ACTION A_ResetFault:
// Sadece arızaları temizle
stHMI.stStatus.bFaultActive := FALSE;
stHMI.stStatus.eFaultCode := E_DisconnectorFault.NONE;
stHMI.stStatus.wsStatusText := "";  // Status text'i temizle

// Timer'ları resetle
tonMotionTimeout(IN := FALSE);
tonContactorOn(IN := FALSE);
tonContactorOff(IN := FALSE);
END_ACTION

ACTION A_ResetStatistics:
// Sadece istatistikleri sıfırla
stHMI.stStatistics.dwOnCount := 0;
stHMI.stStatistics.dwOffCount := 0;
stHMI.stStatistics.dwOperationCount := 0;
stHMI.stStatistics.dwTotalFaultCount := 0;
stHMI.stStatistics.dwThermalFaultCount := 0;
stHMI.stStatistics.dwMotionTimeoutCount := 0;
stHMI.stStatistics.dwContactorFaultCount := 0;
stHMI.stStatistics.dwInterlockFaultCount := 0;
stHMI.stStatistics.tMaxOnTransitionTime := T#0S;
stHMI.stStatistics.tMaxOffTransitionTime := T#0S;
stHMI.stStatistics.tLastOnTransitionTime := T#0S;
stHMI.stStatistics.tLastOffTransitionTime := T#0S;
stHMI.stStatistics.bNewOperationFlag := FALSE;

// Bakım sayacını sıfırla ve operasyon limitini yeniden yükle
stHMI.stStatistics.dwRemainingOperations := stHMI.stConfig.dwOperationLimit;
stHMI.stStatistics.bMaintenanceRequired := FALSE;
END_ACTION

ACTION A_StateMachine:
// Önceki durumu sakla
ePositionPrevious := ePosition;

// Interlock kontrolü
IF bInterlock THEN
    bOnRequest := FALSE;
    bOffRequest := FALSE;
END_IF

// Sürekli pozisyon kontrolü
IF bLimitOn AND bLimitOff THEN
    // Her iki limit aktif - arıza
    ePosition := E_DisconnectorPosition.FAULT;
    stHMI.stStatus.eFaultCode := E_DisconnectorFault.BOTH_LIMITS;
END_IF

// Durum makinesi
CASE ePosition OF
    E_DisconnectorPosition.UNDEFINED:
        // Pozisyon belirleme
        IF bLimitOn AND NOT bLimitOff THEN
            ePosition := E_DisconnectorPosition.ON;
        ELSIF bLimitOff AND NOT bLimitOn THEN
            ePosition := E_DisconnectorPosition.OFF;
        ELSE
            // Ara konumda - komut bekle
            IF bOnRequest THEN
                ePosition := E_DisconnectorPosition.TURNING_ON;
                tOperationStartTime := TIME();
            ELSIF bOffRequest THEN
                ePosition := E_DisconnectorPosition.TURNING_OFF;
                tOperationStartTime := TIME();
            END_IF
        END_IF
        
    E_DisconnectorPosition.OFF:
        // OFF konumunda toprak bıçağı kontrolü
        IF stHMI.stConfig.bEarthSwitchExists AND stHMI.stConfig.bGrounded AND NOT bEarthSwitchOn THEN
            ePosition := E_DisconnectorPosition.FAULT;
            stHMI.stStatus.eFaultCode := E_DisconnectorFault.EARTH_SWITCH;
        END_IF
        
        // ON komutu kontrolü
        IF bOnRequest AND NOT stHMI.stStatus.bFaultActive THEN
            ePosition := E_DisconnectorPosition.TURNING_ON;
            tOperationStartTime := TIME();
        END_IF
        
    E_DisconnectorPosition.TURNING_ON:
        // STOP komutu veya ters yön komutu
        IF stHMI.stCommand.bStop OR bOffRequest THEN
            ePosition := E_DisconnectorPosition.UNDEFINED;
        END_IF
        
        // ON'a ulaşma kontrolü
        IF bLimitOn THEN
            ePosition := E_DisconnectorPosition.ON;
            // İstatistik güncelle
            stHMI.stStatistics.dwOnCount := stHMI.stStatistics.dwOnCount + 1;
            stHMI.stStatistics.tLastOnTransitionTime := TIME() - tOperationStartTime;
            
            // ON konumuna ulaştığında toprak bıçağı kontrolü
            IF stHMI.stConfig.bEarthSwitchExists AND stHMI.stConfig.bGrounded AND NOT bEarthSwitchOff THEN
                ePosition := E_DisconnectorPosition.FAULT;
                stHMI.stStatus.eFaultCode := E_DisconnectorFault.EARTH_SWITCH;
            END_IF
        END_IF
        
    E_DisconnectorPosition.ON:
        // ON konumunda toprak bıçağı kontrolü
        IF stHMI.stConfig.bEarthSwitchExists AND stHMI.stConfig.bGrounded AND NOT bEarthSwitchOff THEN
            ePosition := E_DisconnectorPosition.FAULT;
            stHMI.stStatus.eFaultCode := E_DisconnectorFault.EARTH_SWITCH;
        END_IF
        
        // OFF komutu kontrolü
        IF bOffRequest AND NOT stHMI.stStatus.bFaultActive THEN
            ePosition := E_DisconnectorPosition.TURNING_OFF;
            tOperationStartTime := TIME();
        END_IF
        
    E_DisconnectorPosition.TURNING_OFF:
        // STOP komutu veya ters yön komutu
        IF stHMI.stCommand.bStop OR bOnRequest THEN
            ePosition := E_DisconnectorPosition.UNDEFINED;
        END_IF
        
        // OFF'a ulaşma kontrolü
        IF bLimitOff THEN
            ePosition := E_DisconnectorPosition.OFF;
            // İstatistik güncelle
            stHMI.stStatistics.dwOffCount := stHMI.stStatistics.dwOffCount + 1;
            stHMI.stStatistics.tLastOffTransitionTime := TIME() - tOperationStartTime;
            
            // OFF konumuna ulaştığında toprak bıçağı kontrolü
            IF stHMI.stConfig.bEarthSwitchExists AND stHMI.stConfig.bGrounded AND NOT bEarthSwitchOn THEN
                ePosition := E_DisconnectorPosition.FAULT;
                stHMI.stStatus.eFaultCode := E_DisconnectorFault.EARTH_SWITCH;
            END_IF
        END_IF
        
    E_DisconnectorPosition.FAULT:
        // Arıza durumunda reset bekle
        IF rtrigResetFault.Q THEN
            ePosition := E_DisconnectorPosition.UNDEFINED;
        END_IF
END_CASE
END_ACTION

ACTION A_UpdateStatus:
// PLC Kontrol Durumu
stHMI.stStatus.bPLCControlActive := bPLCControl;

// Aktif Kontrol Modu
stHMI.stStatus.eActiveMode := stHMI.stCommand.eControlMode;

// Pozisyon bilgisini güncelle
stHMI.stStatus.ePosition := ePosition;

// Toprak bıçağı pozisyonunu status'e kopyala
stHMI.stStatus.eEarthSwitchPosition := eEarthSwitchPosition;

// Hareket durumları
stHMI.stStatus.bTurningOn := (ePosition = E_DisconnectorPosition.TURNING_ON);
stHMI.stStatus.bTurningOff := (ePosition = E_DisconnectorPosition.TURNING_OFF);

// Kontaktör çıkışlarını status'e kopyala
stHMI.stStatus.bContactorOn_Out := bContactorOn_Out;
stHMI.stStatus.bContactorOff_Out := bContactorOff_Out;

// Operasyonel durum belirleme
IF stHMI.stStatus.bFaultActive THEN
    stHMI.stStatus.eStatus := E_DisconnectorStatus.FAULTED;
ELSIF NOT bPLCControl THEN
    stHMI.stStatus.eStatus := E_DisconnectorStatus.NO_CONTROL;
ELSIF bInterlock THEN
    stHMI.stStatus.eStatus := E_DisconnectorStatus.INTERLOCKED;
ELSIF stHMI.stStatus.bTurningOn OR stHMI.stStatus.bTurningOff THEN
    stHMI.stStatus.eStatus := E_DisconnectorStatus.OPERATING;
ELSIF stHMI.stStatistics.bMaintenanceRequired THEN
    stHMI.stStatus.eStatus := E_DisconnectorStatus.MAINTENANCE;
ELSE
    stHMI.stStatus.eStatus := E_DisconnectorStatus.READY;
END_IF

// Status text güncelleme
CASE stHMI.stStatus.eStatus OF
    E_DisconnectorStatus.READY:
        CASE ePosition OF
            E_DisconnectorPosition.ON: stHMI.stStatus.wsStatusText := "Hazır - ON pozisyonunda";
            E_DisconnectorPosition.OFF: stHMI.stStatus.wsStatusText := "Hazır - OFF pozisyonunda";
            E_DisconnectorPosition.UNDEFINED: stHMI.stStatus.wsStatusText := "Hazır - Pozisyon belirsiz";
        END_CASE
        
    E_DisconnectorStatus.OPERATING:
        IF stHMI.stStatus.bTurningOn THEN
            stHMI.stStatus.wsStatusText := "ON pozisyonuna gidiyor";
        ELSE
            stHMI.stStatus.wsStatusText := "OFF pozisyonuna gidiyor";
        END_IF
        
    E_DisconnectorStatus.INTERLOCKED:
        stHMI.stStatus.wsStatusText := "Interlock aktif - Komut bekliyor";
        
    E_DisconnectorStatus.NO_CONTROL:
        stHMI.stStatus.wsStatusText := "PLC kontrolü yok - Remote modda";
        
    E_DisconnectorStatus.MAINTENANCE:
        stHMI.stStatus.wsStatusText := "Bakım gerekli!";
END_CASE
END_ACTION

METHOD M_OutputControl : BOOL
VAR_INPUT
    Reset: BOOL;
    Invert: BOOL;
    Momentary: BOOL;
    Set: BOOL;
END_VAR
VAR_OUTPUT
    Out: BOOL;
END_VAR
VAR
    ActiveMode: INT;
    OutLast: BOOL;
END_VAR
IF Reset THEN
    ActiveMode := 0;
ELSIF Invert THEN
    ActiveMode := 1;
ELSIF Momentary THEN
    ActiveMode := 2;
ELSIF Set THEN
    ActiveMode := 3;    
END_IF

CASE ActiveMode OF
    0: //RESET
        Out := FALSE;
        
    1: // INVERT
        IF Invert AND NOT OutLast THEN
            Out := NOT Out;
        END_IF    
        
        OutLast := Invert;    
                    
    2: //PUSH BUTTON (MOMENTARY)
        IF Momentary THEN
            Out := TRUE;
        ELSE
            Out := FALSE;
        END_IF
    3: // SET
        IF Set THEN
            Out := TRUE;
        END_IF    
END_CASE

M_OutputControl := TRUE;
END_METHOD

END_FUNCTION_BLOCK

// ---- POUs/Example/PRG_ContactorExample.TcPOU
PROGRAM PRG_ContactorExample
VAR
    // Function Block Instance
    fbContactor1: FB_ContactorControl;
    
    // Başlangıç konfigürasyonu için flag
    bInitDone: BOOL;
END_VAR


// İlk çalıştırma konfigürasyonu
IF NOT bInitDone THEN
    // Konfigürasyon parametreleri
    GVL_HMI.stContactor1_HMI.stConfig.sProjectCode := '+EP1-K1';
    GVL_HMI.stContactor1_HMI.stConfig.sProductCode := 'ABB A30-30-10 30A';
    GVL_HMI.stContactor1_HMI.stConfig.rRatedCurrent := 30.0;
    GVL_HMI.stContactor1_HMI.stConfig.rRatedVoltage := 400.0;
    GVL_HMI.stContactor1_HMI.stConfig.nPhaseCount := 3;
    GVL_HMI.stContactor1_HMI.stConfig.tFeedbackDelay := T#500MS;
    GVL_HMI.stContactor1_HMI.stConfig.tWeldedDelay := T#2S;
    GVL_HMI.stContactor1_HMI.stConfig.dwOperationLimit := 100000;
    
    // Başlangıç bakım sayacı
    GVL_HMI.stContactor1_HMI.stStatistics.dwRemainingOperations := GVL_HMI.stContactor1_HMI.stConfig.dwOperationLimit;
    
    bInitDone := TRUE;
END_IF

// Function Block Çağrısı
fbContactor1(
    // Fiziksel Girişler
    bFeedback := stContactor1_IO.bFeedback,
    bPLCControl := stContactor1_IO.bPLCControl,
    
    // Güvenlik Girişleri
    bSafetyLoop := GVL_Safety.bSafetyLoop,
    bInterlock := GVL_Safety.bContactor1_Interlock,
    
    // Sistem Girişleri
    bMasterReset := GVL_System.bMasterReset,
    
    // HMI Bağlantısı
    stHMI := GVL_HMI.stContactor1_HMI,
    
    // Fiziksel Çıkış
    bOutput => stContactor1_IO.bOutput
);

// SQL Kayıt İşlemi
IF GVL_HMI.stContactor1_HMI.stStatistics.bNewOperationFlag THEN
    // SQL kayıt fonksiyonunu çağır
    GVL_HMI.stContactor1_HMI.stStatistics.bNewOperationFlag := FALSE;
END_IF

END_PROGRAM

// ---- _ES/12_Contactor/FB_ContactorControl.TcPOU
FUNCTION_BLOCK FB_ContactorControl
VAR_INPUT
    // Fiziksel Girişler
    bFeedback: BOOL;                            // Kontaktör yardımcı kontak geri bildirimi
    bPLCControl: BOOL;                          // PLC kontrol seçici
    
    // Güvenlik Girişleri
    bSafetyLoop: BOOL;                          // Safety loop
    bInterlock: BOOL;                           // Dış interlock sinyali
    
    // Sistem Girişleri
    bMasterReset: BOOL;                         // Master reset
END_VAR

VAR_OUTPUT
    // Fiziksel Çıkış
    bOutput: BOOL;                              // Kontaktör bobini
END_VAR

VAR_IN_OUT
    stHMI: ST_ContactorHMI;                     // HMI için tüm veriler
END_VAR

VAR
    // Position Machine
    ePosition: E_ContactorPosition;             // İç pozisyon değişkeni
    ePositionPrevious: E_ContactorPosition;     // Önceki pozisyon
    
    // Timer'lar
    tonFeedbackOn: TON;                         // ON geri bildirim timer'ı
    tonFeedbackOff: TON;                        // OFF geri bildirim timer'ı
    tonWeldedCheck: TON;                        // Yapışma kontrol timer'ı
    
    // Edge Detection
    rtrigOnCmd: R_TRIG;                         // ON komut yükselen kenar
    rtrigOffCmd: R_TRIG;                        // OFF komut yükselen kenar
    rtrigResetFault: R_TRIG;                    // Reset yükselen kenar
    rtrigResetStatistics: R_TRIG;               // İstatistik reset yükselen kenar
    rtrigMasterReset: R_TRIG;                   // Master reset yükselen kenar
    
    // İç Değişkenler
    bOnRequest: BOOL;                           // Dahili ON isteği
    bOffRequest: BOOL;                          // Dahili OFF isteği
    bBlock: BOOL;                               // Hareket blokaj
END_VAR

// Edge Detection
rtrigOnCmd(CLK := bOnRequest);
rtrigOffCmd(CLK := bOffRequest);
rtrigResetFault(CLK := stHMI.stCommand.bResetFault OR bMasterReset);
rtrigResetStatistics(CLK := stHMI.stCommand.bResetStatistics);
rtrigMasterReset(CLK := bMasterReset);

// Reset İşlemleri
IF rtrigResetFault.Q THEN
    A_ResetFault();
END_IF

IF rtrigResetStatistics.Q OR rtrigMasterReset.Q THEN
    A_ResetStatistics();
END_IF

// Ana kontrol akışı
A_ModeSelection();      // Mod seçimi ve komut belirleme
A_PositionCheck();      // Pozisyon güncelleme
A_FaultCheck();         // Arıza kontrolü
A_Control();            // Çıkış kontrolü
A_UpdateStatus();       // Status güncelleme

// Önceki pozisyonu sakla
ePositionPrevious := ePosition;

ACTION A_Control:
// Blokaj şartları
bBlock := 	bInterlock OR 
          	stHMI.stStatus.bFaultActive OR 
          	NOT bSafetyLoop OR
			bOffRequest;

// Kontaktör kontrolü - Set/Reset mantığı ile
M_OutputControl(
    Invert      := FALSE, 
    Momentary   := FALSE, 
    Set         := bOnRequest,
    Reset       := bBlock,  
    Out         => bOutput
);

// Çıkışı status'e kopyala
stHMI.stStatus.bOutput := bOutput;
END_ACTION

ACTION A_FaultCheck:
// Geri bildirim kontrolü (eğer gerekli ise)
IF stHMI.stConfig.bFeedbackRequired THEN
    // ON geri besleme kontrolü - çıkış var ama geri besleme yok
    tonFeedbackOn(IN := bOutput AND NOT bFeedback, PT := stHMI.stConfig.tFeedbackDelay);
    IF tonFeedbackOn.Q THEN
        stHMI.stStatus.bFaultActive := TRUE;
        stHMI.stStatus.eFaultCode := E_ContactorFault.FEEDBACK;
        stHMI.stStatus.wsStatusText := "ARIZA: Kontaktör ON geri besleme hatası";
    END_IF

    // OFF geri besleme kontrolü - çıkış yok ama geri besleme var (yapışma)
    tonFeedbackOff(IN := NOT bOutput AND bFeedback, PT := stHMI.stConfig.tFeedbackDelay);
    IF tonFeedbackOff.Q THEN
        // Daha uzun süre kontrol et - gerçekten yapışma mı?
        tonWeldedCheck(IN := TRUE, PT := stHMI.stConfig.tWeldedDelay);
        IF tonWeldedCheck.Q THEN
            stHMI.stStatus.bFaultActive := TRUE;
            stHMI.stStatus.eFaultCode := E_ContactorFault.WELDED;
            stHMI.stStatus.wsStatusText := "ARIZA: Kontaktör kontakları yapışmış";
        END_IF
    ELSE
        tonWeldedCheck(IN := FALSE);
    END_IF
ELSE
    // Geri bildirim kontrolü yapılmıyor - timer'ları resetle
    tonFeedbackOn(IN := FALSE);
    tonFeedbackOff(IN := FALSE);
    tonWeldedCheck(IN := FALSE);
END_IF
END_ACTION

ACTION A_ModeSelection:
// PLC kontrolü yoksa mod otomatik olarak REMOTE olur
IF NOT bPLCControl THEN
    stHMI.stStatus.eActiveMode := E_ContactorControlMode.REMOTE;
    bOnRequest := FALSE;
    bOffRequest := FALSE;
    stHMI.stCommand.bManualOnCmd := FALSE;
    stHMI.stCommand.bManualOffCmd := FALSE;
    RETURN;
END_IF

// PLC kontrolü varsa komut edilen modu kullan
IF stHMI.stCommand.eControlMode = E_ContactorControlMode.REMOTE THEN
    stHMI.stStatus.eActiveMode := E_ContactorControlMode.AUTO;
ELSE
    stHMI.stStatus.eActiveMode := stHMI.stCommand.eControlMode;
END_IF

// Kontrol moduna göre komut seçimi
CASE stHMI.stStatus.eActiveMode OF
    E_ContactorControlMode.MANUAL:
        bOnRequest := stHMI.stCommand.bManualOnCmd;
        bOffRequest := stHMI.stCommand.bManualOffCmd;
        
    E_ContactorControlMode.AUTO:
        bOnRequest := stHMI.stCommand.bAutoOnCmd;
        bOffRequest := stHMI.stCommand.bAutoOffCmd;
        
    E_ContactorControlMode.REMOTE:
        bOnRequest := stHMI.stCommand.bManualOnCmd;
        bOffRequest := stHMI.stCommand.bManualOffCmd;
END_CASE

// Çift komut kontrolü
IF bOnRequest AND bOffRequest THEN
    bOnRequest := FALSE;
    bOffRequest := FALSE;
END_IF
END_ACTION

ACTION A_PositionCheck:
// Kontaktör pozisyon kontrolü
IF stHMI.stConfig.bFeedbackRequired THEN
    // Geri bildirim varsa kullan
    IF bOutput AND bFeedback THEN
        ePosition := E_ContactorPosition.ON;
    ELSIF NOT bOutput AND NOT bFeedback THEN
        ePosition := E_ContactorPosition.OFF;
    ELSE
        // Çıkış var ama geri besleme yok veya tam tersi
        ePosition := E_ContactorPosition.UNDEFINED;
    END_IF
ELSE
    // Geri bildirim yoksa sadece çıkışa göre pozisyon belirle
    IF bOutput THEN
        ePosition := E_ContactorPosition.ON;
    ELSE
        ePosition := E_ContactorPosition.OFF;
    END_IF
END_IF
END_ACTION

ACTION A_ResetFault:
// Arızaları temizle
stHMI.stStatus.bFaultActive := FALSE;
stHMI.stStatus.eFaultCode := E_ContactorFault.NONE;
stHMI.stStatus.wsStatusText := "";

// Timer'ları resetle
tonFeedbackOn(IN := FALSE);
tonFeedbackOff(IN := FALSE);
tonWeldedCheck(IN := FALSE);
END_ACTION

ACTION A_ResetStatistics:
// İstatistikleri sıfırla
stHMI.stStatistics.dwOnCount := 0;
stHMI.stStatistics.dwOffCount := 0;
stHMI.stStatistics.dwOperationCount := 0;
stHMI.stStatistics.dwTotalFaultCount := 0;
stHMI.stStatistics.dwFeedbackFaultCount := 0;
stHMI.stStatistics.dwWeldedFaultCount := 0;
stHMI.stStatistics.bNewOperationFlag := FALSE;

// Bakım sayacını sıfırla ve operasyon limitini yeniden yükle
stHMI.stStatistics.dwRemainingOperations := stHMI.stConfig.dwOperationLimit;
stHMI.stStatistics.bMaintenanceRequired := FALSE;
END_ACTION

ACTION A_UpdateStatus:
// PLC Kontrol Durumu
stHMI.stStatus.bPLCControlActive := bPLCControl;

// Aktif Kontrol Modu
stHMI.stStatus.eActiveMode := stHMI.stCommand.eControlMode;

// Pozisyon bilgisini güncelle
stHMI.stStatus.ePosition := ePosition;

// Operasyonel durum belirleme
IF stHMI.stStatus.bFaultActive THEN
    stHMI.stStatus.eStatus := E_ContactorStatus.FAULTED;
ELSIF NOT bPLCControl THEN
    stHMI.stStatus.eStatus := E_ContactorStatus.NO_CONTROL;
ELSIF bInterlock THEN
    stHMI.stStatus.eStatus := E_ContactorStatus.INTERLOCKED;
ELSIF stHMI.stStatistics.bMaintenanceRequired THEN
    stHMI.stStatus.eStatus := E_ContactorStatus.MAINTENANCE;
ELSE
    stHMI.stStatus.eStatus := E_ContactorStatus.READY;
END_IF

// Status text güncelleme
CASE stHMI.stStatus.eStatus OF
    E_ContactorStatus.READY:
        CASE ePosition OF
            E_ContactorPosition.ON: 
                stHMI.stStatus.wsStatusText := "Hazır - Kontaktör ON";
            E_ContactorPosition.OFF: 
                stHMI.stStatus.wsStatusText := "Hazır - Kontaktör OFF";
            E_ContactorPosition.UNDEFINED: 
                stHMI.stStatus.wsStatusText := "Hazır - Durum belirsiz";
        END_CASE
        
    E_ContactorStatus.INTERLOCKED:
        stHMI.stStatus.wsStatusText := "Interlock aktif - Komut bekliyor";
        
    E_ContactorStatus.NO_CONTROL:
        stHMI.stStatus.wsStatusText := "PLC kontrolü yok - Remote modda";
        
    E_ContactorStatus.MAINTENANCE:
        stHMI.stStatus.wsStatusText := "Bakım gerekli!";
        
    E_ContactorStatus.FAULTED:
        ; // Arıza durumunda text zaten A_FaultCheck'te set ediliyor
END_CASE

// İstatistik güncelleme - pozisyon değişiminde
IF ePosition <> ePositionPrevious THEN
    IF ePosition = E_ContactorPosition.ON THEN
        stHMI.stStatistics.dwOnCount := stHMI.stStatistics.dwOnCount + 1;
        stHMI.stStatistics.dwOperationCount := stHMI.stStatistics.dwOperationCount + 1;
    ELSIF ePosition = E_ContactorPosition.OFF AND ePositionPrevious = E_ContactorPosition.ON THEN
        stHMI.stStatistics.dwOffCount := stHMI.stStatistics.dwOffCount + 1;
        stHMI.stStatistics.dwOperationCount := stHMI.stStatistics.dwOperationCount + 1;
    END_IF
    
    // Bakım kontrolü
    stHMI.stStatistics.dwRemainingOperations := stHMI.stConfig.dwOperationLimit - stHMI.stStatistics.dwOperationCount;
    IF stHMI.stStatistics.dwRemainingOperations < 1000 THEN
        stHMI.stStatistics.bMaintenanceRequired := TRUE;
    END_IF
END_IF
END_ACTION

METHOD M_OutputControl : BOOL
VAR_INPUT
    Reset: BOOL;
    Invert: BOOL;
    Momentary: BOOL;
    Set: BOOL;
END_VAR
VAR_OUTPUT
    Out: BOOL;
END_VAR
VAR
    ActiveMode: INT;
    OutLast: BOOL;
END_VAR
IF Reset THEN
    ActiveMode := 0;
ELSIF Invert THEN
    ActiveMode := 1;
ELSIF Momentary THEN
    ActiveMode := 2;
ELSIF Set THEN
    ActiveMode := 3;    
END_IF

CASE ActiveMode OF
    0: //RESET
        Out := FALSE;
        
    1: // INVERT
        IF Invert AND NOT OutLast THEN
            Out := NOT Out;
        END_IF    
        
        OutLast := Invert;    
                    
    2: //PUSH BUTTON (MOMENTARY)
        IF Momentary THEN
            Out := TRUE;
        ELSE
            Out := FALSE;
        END_IF
    3: // SET
        IF Set THEN
            Out := TRUE;
        END_IF    
END_CASE

M_OutputControl := TRUE;
END_METHOD

END_FUNCTION_BLOCK

// ---- POUs/Example/PRG_CircuitBreakerExample.TcPOU
PROGRAM PRG_CircuitBreakerExample
VAR
    // Function Block Instance
    fbCircuitBreaker1: FB_CircuitBreaker;
    
    // Başlangıç konfigürasyonu için flag
    bInitDone: BOOL;
END_VAR


// İlk çalıştırma konfigürasyonu
IF NOT bInitDone THEN
    // Konfigürasyon parametreleri
    GVL_HMI.stCircuitBreaker1_HMI.stConfig.sProjectCode := '+EP1-Q1';
    GVL_HMI.stCircuitBreaker1_HMI.stConfig.sProductCode := 'ABB VD4 1250A';
    GVL_HMI.stCircuitBreaker1_HMI.stConfig.rRatedCurrent := 1250.0;
    GVL_HMI.stCircuitBreaker1_HMI.stConfig.rRatedVoltage := 12.0;
    GVL_HMI.stCircuitBreaker1_HMI.stConfig.nPhaseCount := 3;
    GVL_HMI.stCircuitBreaker1_HMI.stConfig.tMotionTimeout := T#5S;
    GVL_HMI.stCircuitBreaker1_HMI.stConfig.tSpringChargeTimeout := T#30S;
    GVL_HMI.stCircuitBreaker1_HMI.stConfig.bSpringChargeRequired := TRUE;
    GVL_HMI.stCircuitBreaker1_HMI.stConfig.dwOperationLimit := 10000;
    
    // Başlangıç bakım sayacı
    GVL_HMI.stCircuitBreaker1_HMI.stStatistics.dwRemainingOperations := GVL_HMI.stCircuitBreaker1_HMI.stConfig.dwOperationLimit;
    
    bInitDone := TRUE;
END_IF

// Function Block Çağrısı
fbCircuitBreaker1(
    // Fiziksel Girişler
    bPositionOn := stCircuitBreaker1_IO.bPositionOn,
    bPositionOff := stCircuitBreaker1_IO.bPositionOff,
    bPositionTripped := stCircuitBreaker1_IO.bPositionTripped,
    bSpringCharged := stCircuitBreaker1_IO.bSpringCharged,
    bPLCControl := stCircuitBreaker1_IO.bPLCControl,
    
    // Güvenlik Girişleri
    bSafetyLoop := GVL_Safety.bSafetyLoop,
    bInterlock := GVL_Safety.bCircuitBreaker1_Interlock,
    
    // Sistem Girişleri
    bMasterReset := GVL_System.bMasterReset,
    
    // HMI Bağlantısı
    stHMI := GVL_HMI.stCircuitBreaker1_HMI,
    
    // Fiziksel Çıkışlar
    bOnCommand => stCircuitBreaker1_IO.bOnCommand,
    bOffCommand => stCircuitBreaker1_IO.bOffCommand
);

// SQL Kayıt İşlemi
IF GVL_HMI.stCircuitBreaker1_HMI.stStatistics.bNewOperationFlag THEN
    // SQL kayıt fonksiyonunu çağır
    GVL_HMI.stCircuitBreaker1_HMI.stStatistics.bNewOperationFlag := FALSE;
END_IF

END_PROGRAM

// ---- _ES/13_CircuitBreaker/FB_CircuitBreaker.TcPOU
FUNCTION_BLOCK FB_CircuitBreaker
VAR_INPUT
    // Fiziksel Girişler
    bPositionOn: BOOL;                          // ON pozisyon geri bildirimi
    bPositionOff: BOOL;                         // OFF pozisyon geri bildirimi
    bPositionTripped: BOOL;                     // TRIP pozisyon geri bildirimi
    bSpringCharged: BOOL;                       // Yay kurulu bilgisi
    bPLCControl: BOOL;                          // PLC kontrol seçici
    
    // Güvenlik Girişleri
    bSafetyLoop: BOOL;                          // Safety loop
    bInterlock: BOOL;                           // Dış interlock sinyali
    
    // Sistem Girişleri
    bMasterReset: BOOL;                         // Master reset
END_VAR

VAR_OUTPUT
    // Fiziksel Çıkışlar
    bOnCommand: BOOL;                           // ON komutu
    bOffCommand: BOOL;                          // OFF komutu
END_VAR

VAR_IN_OUT
    stHMI: ST_CircuitBreakerHMI;               // HMI için tüm veriler
END_VAR

VAR
    // Position Machine
    ePosition: E_CircuitBreakerPosition;        // İç pozisyon değişkeni
    ePositionPrevious: E_CircuitBreakerPosition; // Önceki pozisyon
    
    // Timer'lar
    tonMotionTimeout: TON;                      // Hareket zaman aşımı timer'ı
    tonSpringChargeTimeout: TON;                // Yay kurma zaman aşımı timer'ı
    
    // Edge Detection
    rtrigOnCmd: R_TRIG;                         // ON komut yükselen kenar
    rtrigOffCmd: R_TRIG;                        // OFF komut yükselen kenar
    rtrigResetTrip: R_TRIG;                     // Trip reset yükselen kenar
    rtrigResetFault: R_TRIG;                    // Reset yükselen kenar
    rtrigResetStatistics: R_TRIG;               // İstatistik reset yükselen kenar
    rtrigMasterReset: R_TRIG;                   // Master reset yükselen kenar
    
    // İç Değişkenler
    bOnRequest: BOOL;                           // Dahili ON isteği
    bOffRequest: BOOL;                          // Dahili OFF isteği
    bBlockOn: BOOL;                             // ON hareketi blokaj
    bBlockOff: BOOL;                            // OFF hareketi blokaj
    tOperationStartTime: TIME;                  // Operasyon başlangıç zamanı
END_VAR

// Edge Detection
rtrigOnCmd(CLK := bOnRequest);
rtrigOffCmd(CLK := bOffRequest);
rtrigResetTrip(CLK := stHMI.stCommand.bResetTrip);
rtrigResetFault(CLK := stHMI.stCommand.bResetFault OR bMasterReset);
rtrigResetStatistics(CLK := stHMI.stCommand.bResetStatistics);
rtrigMasterReset(CLK := bMasterReset);

// Reset İşlemleri
IF rtrigResetFault.Q OR rtrigResetTrip.Q THEN
    A_ResetFault();
END_IF

IF rtrigResetStatistics.Q OR rtrigMasterReset.Q THEN
    A_ResetStatistics();
END_IF

// Ana kontrol akışı
A_ModeSelection();      // Mod seçimi ve komut belirleme
A_PositionCheck();      // Pozisyon güncelleme
A_FaultCheck();         // Arıza kontrolü
A_Control();            // Çıkış kontrolü
A_UpdateStatus();       // Status güncelleme

// Önceki pozisyonu sakla
ePositionPrevious := ePosition;

// Operasyon zamanı hesaplama
IF (bOnCommand OR bOffCommand) AND tOperationStartTime = T#0S THEN
    tOperationStartTime := TIME();
ELSIF NOT (bOnCommand OR bOffCommand) AND tOperationStartTime > T#0S THEN
    // Operasyon tamamlandı
    tOperationStartTime := T#0S;
END_IF

ACTION A_Control:
// ON hareketi blokaj şartları
bBlockOn := bInterlock OR 
            stHMI.stStatus.bFaultActive OR 
            NOT bSafetyLoop OR
            (ePosition = E_CircuitBreakerPosition.ON) OR
            (ePosition = E_CircuitBreakerPosition.TRIPPED) OR
            (stHMI.stConfig.bSpringChargeRequired AND NOT bSpringCharged);

// OFF hareketi blokaj şartları            
bBlockOff := bInterlock OR 
             stHMI.stStatus.bFaultActive OR 
             NOT bSafetyLoop OR
             (ePosition = E_CircuitBreakerPosition.OFF) OR
             (ePosition = E_CircuitBreakerPosition.TRIPPED);

// ON komutu kontrolü
M_OutputControl(
    Invert      := FALSE, 
    Momentary   := bOnRequest, 
    Set         := FALSE,
    Reset       := bBlockOn OR bOffRequest,  
    Out         => bOnCommand
);

// OFF komutu kontrolü  
M_OutputControl(
    Invert      := FALSE, 
    Momentary   := bOffRequest, 
    Set         := FALSE,
    Reset       := bBlockOff OR bOnRequest,  
    Out         => bOffCommand
);

// Çıkışları status'e kopyala
stHMI.stStatus.bOnCommand := bOnCommand;
stHMI.stStatus.bOffCommand := bOffCommand;
END_ACTION

ACTION A_FaultCheck:
// Birden fazla pozisyon aktif - sensör hatası
IF bPositionOn AND bPositionOff AND NOT bPositionTripped THEN
    stHMI.stStatus.bFaultActive := TRUE;
    stHMI.stStatus.eFaultCode := E_CircuitBreakerFault.FEEDBACK;
    stHMI.stStatus.wsStatusText := "ARIZA: ON ve OFF pozisyonları aynı anda aktif";
    
ELSIF bPositionOn AND bPositionTripped AND NOT bPositionOff THEN
    stHMI.stStatus.bFaultActive := TRUE;
    stHMI.stStatus.eFaultCode := E_CircuitBreakerFault.FEEDBACK;
    stHMI.stStatus.wsStatusText := "ARIZA: ON ve TRIP pozisyonları aynı anda aktif";
    
ELSIF bPositionOff AND bPositionTripped AND NOT bPositionOn THEN
    stHMI.stStatus.bFaultActive := TRUE;
    stHMI.stStatus.eFaultCode := E_CircuitBreakerFault.FEEDBACK;
    stHMI.stStatus.wsStatusText := "ARIZA: OFF ve TRIP pozisyonları aynı anda aktif";
    
ELSIF bPositionOn AND bPositionOff AND bPositionTripped THEN
    stHMI.stStatus.bFaultActive := TRUE;
    stHMI.stStatus.eFaultCode := E_CircuitBreakerFault.FEEDBACK;
    stHMI.stStatus.wsStatusText := "ARIZA: Tüm pozisyonlar aynı anda aktif";
END_IF

// TRIP durumu kontrolü
IF ePosition = E_CircuitBreakerPosition.TRIPPED THEN
    // TRIP durumunda - bu bir arıza değil ama özel durum
    stHMI.stStatus.eStatus := E_CircuitBreakerStatus.TRIPPED;
    stHMI.stStatus.wsStatusText := "DİKKAT: Kesici TRIP pozisyonunda";
    // TRIP durumunda komutları blokla
    bOnRequest := FALSE;
    bOffRequest := FALSE;
END_IF

// Hareket zaman aşımı kontrolü
tonMotionTimeout(IN := (bOnCommand OR bOffCommand) AND (ePosition = E_CircuitBreakerPosition.UNDEFINED), 
                 PT := stHMI.stConfig.tMotionTimeout);
IF tonMotionTimeout.Q THEN
    stHMI.stStatus.bFaultActive := TRUE;
    stHMI.stStatus.eFaultCode := E_CircuitBreakerFault.MOTION_TIMEOUT;
    stHMI.stStatus.wsStatusText := "ARIZA: Hareket zaman aşımı";
END_IF

// Yay kurma arızası kontrolü (eğer gerekli ise)
IF stHMI.stConfig.bSpringChargeRequired THEN
    // ON komutu verildi ama yay kurulu değil
    IF bOnRequest AND NOT bSpringCharged AND (ePosition = E_CircuitBreakerPosition.OFF) THEN
        tonSpringChargeTimeout(IN := TRUE, PT := stHMI.stConfig.tSpringChargeTimeout);
        IF tonSpringChargeTimeout.Q THEN
            stHMI.stStatus.bFaultActive := TRUE;
            stHMI.stStatus.eFaultCode := E_CircuitBreakerFault.SPRING_CHARGE;
            stHMI.stStatus.wsStatusText := "ARIZA: Yay kurma hatası";
        END_IF
    ELSE
        tonSpringChargeTimeout(IN := FALSE);
    END_IF
END_IF
END_ACTION

ACTION A_ModeSelection:
// PLC kontrolü yoksa mod otomatik olarak REMOTE olur
IF NOT bPLCControl THEN
    stHMI.stStatus.eActiveMode := E_CircuitBreakerControlMode.REMOTE;
    bOnRequest := FALSE;
    bOffRequest := FALSE;
    stHMI.stCommand.bManualOnCmd := FALSE;
    stHMI.stCommand.bManualOffCmd := FALSE;
    RETURN;
END_IF

// PLC kontrolü varsa komut edilen modu kullan
IF stHMI.stCommand.eControlMode = E_CircuitBreakerControlMode.REMOTE THEN
    stHMI.stStatus.eActiveMode := E_CircuitBreakerControlMode.AUTO;
ELSE
    stHMI.stStatus.eActiveMode := stHMI.stCommand.eControlMode;
END_IF

// Kontrol moduna göre komut seçimi
CASE stHMI.stStatus.eActiveMode OF
    E_CircuitBreakerControlMode.MANUAL:
        bOnRequest := stHMI.stCommand.bManualOnCmd;
        bOffRequest := stHMI.stCommand.bManualOffCmd;
        
    E_CircuitBreakerControlMode.AUTO:
        bOnRequest := stHMI.stCommand.bAutoOnCmd;
        bOffRequest := stHMI.stCommand.bAutoOffCmd;
        
    E_CircuitBreakerControlMode.REMOTE:
        bOnRequest := stHMI.stCommand.bManualOnCmd;
        bOffRequest := stHMI.stCommand.bManualOffCmd;
END_CASE

// Çift komut kontrolü
IF bOnRequest AND bOffRequest THEN
    bOnRequest := FALSE;
    bOffRequest := FALSE;
END_IF
END_ACTION

ACTION A_PositionCheck:
// Kesici pozisyon kontrolü
IF bPositionOn AND NOT bPositionOff AND NOT bPositionTripped THEN
    ePosition := E_CircuitBreakerPosition.ON;
ELSIF bPositionOff AND NOT bPositionOn AND NOT bPositionTripped THEN
    ePosition := E_CircuitBreakerPosition.OFF;
ELSIF bPositionTripped AND NOT bPositionOn AND NOT bPositionOff THEN
    ePosition := E_CircuitBreakerPosition.TRIPPED;
ELSE
    // Birden fazla pozisyon aktif veya hiçbiri aktif değil
    ePosition := E_CircuitBreakerPosition.UNDEFINED;
END_IF

// Yay durumunu status'e kopyala
stHMI.stStatus.bSpringCharged := bSpringCharged;
END_ACTION

ACTION A_ResetFault:
// Arızaları temizle
stHMI.stStatus.bFaultActive := FALSE;
stHMI.stStatus.eFaultCode := E_CircuitBreakerFault.NONE;
stHMI.stStatus.wsStatusText := "";

// Timer'ları resetle
tonMotionTimeout(IN := FALSE);
tonSpringChargeTimeout(IN := FALSE);

// Trip durumunu kontrol et - eğer hala TRIP pozisyonundaysa durumu güncelle
IF bPositionTripped THEN
    ePosition := E_CircuitBreakerPosition.TRIPPED;
    stHMI.stStatus.eStatus := E_CircuitBreakerStatus.TRIPPED;
END_IF
END_ACTION

ACTION A_ResetStatistics:
// İstatistikleri sıfırla
stHMI.stStatistics.dwOnCount := 0;
stHMI.stStatistics.dwOffCount := 0;
stHMI.stStatistics.dwTripCount := 0;
stHMI.stStatistics.dwOperationCount := 0;
stHMI.stStatistics.dwTotalFaultCount := 0;
stHMI.stStatistics.dwSpringChargeFaultCount := 0;
stHMI.stStatistics.dwMotionTimeoutCount := 0;
stHMI.stStatistics.dwTripCoilFaultCount := 0;
stHMI.stStatistics.bNewOperationFlag := FALSE;

// Bakım sayacını sıfırla ve operasyon limitini yeniden yükle
stHMI.stStatistics.dwRemainingOperations := stHMI.stConfig.dwOperationLimit;
stHMI.stStatistics.bMaintenanceRequired := FALSE;
END_ACTION

ACTION A_UpdateStatus:
// PLC Kontrol Durumu
stHMI.stStatus.bPLCControlActive := bPLCControl;

// Aktif Kontrol Modu
stHMI.stStatus.eActiveMode := stHMI.stCommand.eControlMode;

// Pozisyon bilgisini güncelle
stHMI.stStatus.ePosition := ePosition;

// Yay durumu
stHMI.stStatus.bSpringCharged := bSpringCharged;

// Operasyonel durum belirleme
IF stHMI.stStatus.bFaultActive THEN
    stHMI.stStatus.eStatus := E_CircuitBreakerStatus.FAULTED;
ELSIF ePosition = E_CircuitBreakerPosition.TRIPPED THEN
    stHMI.stStatus.eStatus := E_CircuitBreakerStatus.TRIPPED;
ELSIF NOT bPLCControl THEN
    stHMI.stStatus.eStatus := E_CircuitBreakerStatus.NO_CONTROL;
ELSIF bInterlock THEN
    stHMI.stStatus.eStatus := E_CircuitBreakerStatus.INTERLOCKED;
ELSIF bOnCommand OR bOffCommand THEN
    stHMI.stStatus.eStatus := E_CircuitBreakerStatus.OPERATING;
ELSIF stHMI.stStatistics.bMaintenanceRequired THEN
    stHMI.stStatus.eStatus := E_CircuitBreakerStatus.MAINTENANCE;
ELSE
    stHMI.stStatus.eStatus := E_CircuitBreakerStatus.READY;
END_IF

// Status text güncelleme (arıza değilse)
IF NOT stHMI.stStatus.bFaultActive AND (ePosition <> E_CircuitBreakerPosition.TRIPPED) THEN
    CASE stHMI.stStatus.eStatus OF
        E_CircuitBreakerStatus.READY:
            CASE ePosition OF
                E_CircuitBreakerPosition.ON: 
                    stHMI.stStatus.wsStatusText := "Hazır - Kesici ON";
                E_CircuitBreakerPosition.OFF: 
                    IF stHMI.stConfig.bSpringChargeRequired AND NOT bSpringCharged THEN
                        stHMI.stStatus.wsStatusText := "Hazır - Kesici OFF (Yay kurulu değil)";
                    ELSE
                        stHMI.stStatus.wsStatusText := "Hazır - Kesici OFF";
                    END_IF
                E_CircuitBreakerPosition.UNDEFINED: 
                    stHMI.stStatus.wsStatusText := "Hazır - Pozisyon belirsiz";
            END_CASE
            
        E_CircuitBreakerStatus.OPERATING:
            IF bOnCommand THEN
                stHMI.stStatus.wsStatusText := "ON pozisyonuna gidiyor";
            ELSE
                stHMI.stStatus.wsStatusText := "OFF pozisyonuna gidiyor";
            END_IF
            
        E_CircuitBreakerStatus.INTERLOCKED:
            stHMI.stStatus.wsStatusText := "Interlock aktif - Komut bekliyor";
            
        E_CircuitBreakerStatus.NO_CONTROL:
            stHMI.stStatus.wsStatusText := "PLC kontrolü yok - Remote modda";
            
        E_CircuitBreakerStatus.MAINTENANCE:
            stHMI.stStatus.wsStatusText := "Bakım gerekli!";
    END_CASE
END_IF

// İstatistik güncelleme - pozisyon değişiminde
IF ePosition <> ePositionPrevious THEN
    CASE ePosition OF
        E_CircuitBreakerPosition.ON:
            stHMI.stStatistics.dwOnCount := stHMI.stStatistics.dwOnCount + 1;
            stHMI.stStatistics.dwOperationCount := stHMI.stStatistics.dwOperationCount + 1;
            
        E_CircuitBreakerPosition.OFF:
            IF ePositionPrevious = E_CircuitBreakerPosition.ON THEN
                stHMI.stStatistics.dwOffCount := stHMI.stStatistics.dwOffCount + 1;
                stHMI.stStatistics.dwOperationCount := stHMI.stStatistics.dwOperationCount + 1;
            END_IF
            
        E_CircuitBreakerPosition.TRIPPED:
            stHMI.stStatistics.dwTripCount := stHMI.stStatistics.dwTripCount + 1;
    END_CASE
    
    // Bakım kontrolü
    stHMI.stStatistics.dwRemainingOperations := stHMI.stConfig.dwOperationLimit - stHMI.stStatistics.dwOperationCount;
    IF stHMI.stStatistics.dwRemainingOperations < 100 THEN
        stHMI.stStatistics.bMaintenanceRequired := TRUE;
    END_IF
END_IF
END_ACTION

METHOD M_OutputControl : BOOL
VAR_INPUT
    Reset: BOOL;
    Invert: BOOL;
    Momentary: BOOL;
    Set: BOOL;
END_VAR
VAR_OUTPUT
    Out: BOOL;
END_VAR
VAR
    ActiveMode: INT;
    OutLast: BOOL;
END_VAR
IF Reset THEN
    ActiveMode := 0;
ELSIF Invert THEN
    ActiveMode := 1;
ELSIF Momentary THEN
    ActiveMode := 2;
ELSIF Set THEN
    ActiveMode := 3;    
END_IF

CASE ActiveMode OF
    0: //RESET
        Out := FALSE;
        
    1: // INVERT
        IF Invert AND NOT OutLast THEN
            Out := NOT Out;
        END_IF    
        
        OutLast := Invert;    
                    
    2: //PUSH BUTTON (MOMENTARY)
        IF Momentary THEN
            Out := TRUE;
        ELSE
            Out := FALSE;
        END_IF
    3: // SET
        IF Set THEN
            Out := TRUE;
        END_IF    
END_CASE

M_OutputControl := TRUE;
END_METHOD

END_FUNCTION_BLOCK

// ---- POUs/Example/PRG_Simulation.TcPOU
PROGRAM PRG_Simulation
VAR
    // Simülasyon kontrol
    bSimulationEnable: BOOL := TRUE;
    
    // Disconnector simülasyon komutları
    bSimOnCmd: BOOL;
    bSimOffCmd: BOOL;
    bSimThermalFault: BOOL;
    bSimInterlock: BOOL;
    bSimEarthSwitchError: BOOL;
    
    // Contactor simülasyon komutları
    bSimContactor1_OnCmd: BOOL;
    bSimContactor1_OffCmd: BOOL;
    bSimContactor1_FeedbackFault: BOOL;
    bSimContactor1_Welded: BOOL;
    bSimContactor1_Interlock: BOOL;
    
    // Simülasyon parametreleri
    tOnDelay: TIME := T#2S;
    tOffDelay: TIME := T#2S;
    tContactorResponseDelay: TIME := T#200MS;
    tContactorFeedbackDelay: TIME := T#100MS;
	
    // Circuit Breaker simülasyon komutları
    bSimBreaker1_OnCmd: BOOL;
    bSimBreaker1_OffCmd: BOOL;
    bSimBreaker1_Trip: BOOL;
    bSimBreaker1_SpringNotCharged: BOOL;
    bSimBreaker1_Interlock: BOOL;
    
    // Circuit Breaker simülasyon parametreleri
    tBreakerMotionDelay: TIME := T#3S;
END_VAR

// =====================================================
// ANA GÖVDE
// =====================================================

IF bSimulationEnable THEN
    
    // ============= DISCONNECTOR 1 SIMULATION =============
    M_SimulateDisconnector(
        sDisconnectorName := 'Disconnector1',
        i_bSimEnable := TRUE,
        i_bSimThermalFault := bSimThermalFault,
        i_bSimEarthSwitchError := bSimEarthSwitchError,
        i_tOnDelay := tOnDelay,
        i_tOffDelay := tOffDelay,
        i_tContactorDelay := tContactorResponseDelay,
        io_stIO := stDisconnector1_IO
    );
    
    // Disconnector Interlock simülasyonu
    GVL_Safety.bDisconnector1_Interlock := bSimInterlock;
    
    // Disconnector HMI komut simülasyonu
    IF bSimOnCmd THEN
        GVL_HMI.stDisconnector1_HMI.stCommand.bManualOnCmd := TRUE;
        GVL_HMI.stDisconnector1_HMI.stCommand.bManualOffCmd := FALSE;
    ELSIF bSimOffCmd THEN
        GVL_HMI.stDisconnector1_HMI.stCommand.bManualOnCmd := FALSE;
        GVL_HMI.stDisconnector1_HMI.stCommand.bManualOffCmd := TRUE;
    ELSE
        GVL_HMI.stDisconnector1_HMI.stCommand.bManualOnCmd := FALSE;
        GVL_HMI.stDisconnector1_HMI.stCommand.bManualOffCmd := FALSE;
    END_IF
    
    // Disconnector mod seçimi
    GVL_HMI.stDisconnector1_HMI.stCommand.eControlMode := E_DisconnectorControlMode.MANUAL;
    
    // ============= CONTACTOR 1 SIMULATION =============
	M_SimulateContactor(
		sContactorName := 'Contactor1',
		i_bSimEnable := TRUE,
		i_bSimFeedbackFault := bSimContactor1_FeedbackFault,
		i_bSimWelded := bSimContactor1_Welded,
		i_tFeedbackDelay := tContactorFeedbackDelay,
		io_stIO := stContactor1_IO
	);
		
    // Contactor Interlock simülasyonu
    GVL_Safety.bContactor1_Interlock := bSimContactor1_Interlock;
    
    // Contactor HMI komut simülasyonu
    IF bSimContactor1_OnCmd THEN
        GVL_HMI.stContactor1_HMI.stCommand.bManualOnCmd := TRUE;
        GVL_HMI.stContactor1_HMI.stCommand.bManualOffCmd := FALSE;
    ELSIF bSimContactor1_OffCmd THEN
        GVL_HMI.stContactor1_HMI.stCommand.bManualOnCmd := FALSE;
        GVL_HMI.stContactor1_HMI.stCommand.bManualOffCmd := TRUE;
    ELSE
        GVL_HMI.stContactor1_HMI.stCommand.bManualOnCmd := FALSE;
        GVL_HMI.stContactor1_HMI.stCommand.bManualOffCmd := FALSE;
    END_IF
    
    // Contactor mod seçimi
    GVL_HMI.stContactor1_HMI.stCommand.eControlMode := E_ContactorControlMode.MANUAL;
    
    // ============= GENEL SAFETY SIMULATION =============
    // Safety loop simülasyonu (normalde TRUE)
    GVL_Safety.bSafetyLoop := TRUE;
    
    // Master reset simülasyonu
    GVL_System.bMasterReset := FALSE;
    
END_IF

// =====================================================
// DURUM GÖSTERIMI (Debug için)
// =====================================================
// Disconnector Status: GVL_HMI.stDisconnector1_HMI.stStatus.sStatusText
// Disconnector Position: GVL_HMI.stDisconnector1_HMI.stStatus.ePosition
// Disconnector Fault: GVL_HMI.stDisconnector1_HMI.stStatus.eFaultCode
// 
// Contactor Status: GVL_HMI.stContactor1_HMI.stStatus.sStatusText
// Contactor Position: GVL_HMI.stContactor1_HMI.stStatus.ePosition
// Contactor Fault: GVL_HMI.stContactor1_HMI.stStatus.eFaultCode


// ============= CIRCUIT BREAKER 1 SIMULATION =============
    M_SimulateCircuitBreaker(
        sBreakerName := 'CircuitBreaker1',
        i_bSimEnable := TRUE,
        i_bSimTrip := bSimBreaker1_Trip,
        i_bSimSpringNotCharged := bSimBreaker1_SpringNotCharged,
        i_tMotionDelay := tBreakerMotionDelay,
        io_stIO := GVL_IO.stCircuitBreaker1_IO
    );
    
    // Circuit Breaker Interlock simülasyonu
    GVL_Safety.bCircuitBreaker1_Interlock := bSimBreaker1_Interlock;
    
    // Circuit Breaker HMI komut simülasyonu
    IF bSimBreaker1_OnCmd THEN
        GVL_HMI.stCircuitBreaker1_HMI.stCommand.bManualOnCmd := TRUE;
        GVL_HMI.stCircuitBreaker1_HMI.stCommand.bManualOffCmd := FALSE;
    ELSIF bSimBreaker1_OffCmd THEN
        GVL_HMI.stCircuitBreaker1_HMI.stCommand.bManualOnCmd := FALSE;
        GVL_HMI.stCircuitBreaker1_HMI.stCommand.bManualOffCmd := TRUE;
    ELSE
        GVL_HMI.stCircuitBreaker1_HMI.stCommand.bManualOnCmd := FALSE;
        GVL_HMI.stCircuitBreaker1_HMI.stCommand.bManualOffCmd := FALSE;
    END_IF
    
    // Circuit Breaker mod seçimi
    GVL_HMI.stCircuitBreaker1_HMI.stCommand.eControlMode := E_CircuitBreakerControlMode.MANUAL;

METHOD M_SimulateCircuitBreaker : BOOL
VAR_INPUT
    sBreakerName: STRING;                   // Kesici adı
    i_bSimEnable: BOOL;                     // Simülasyon aktif mi?
    i_bSimTrip: BOOL;                       // Trip simülasyonu
    i_bSimSpringNotCharged: BOOL;           // Yay kurulu değil simülasyonu
    i_tMotionDelay: TIME;                   // Hareket gecikmesi
END_VAR
VAR_IN_OUT
    io_stIO: ST_CircuitBreakerIO;           // IO structure
END_VAR
VAR_STAT
    tonOnDelay: TON;                        // ON gecikme timer'ı
    tonOffDelay: TON;                       // OFF gecikme timer'ı
    bLastOnCmd: BOOL;                       // Önceki ON komutu
    bLastOffCmd: BOOL;                      // Önceki OFF komutu
END_VAR

IF NOT i_bSimEnable THEN
    M_SimulateCircuitBreaker := FALSE;
    RETURN;
END_IF

// Trip simülasyonu - öncelikli
IF i_bSimTrip THEN
    io_stIO.bPositionOn := FALSE;
    io_stIO.bPositionOff := FALSE;
    io_stIO.bPositionTripped := TRUE;
ELSE
    // Normal pozisyon simülasyonu
    // ON komutu yükselen kenar
    IF io_stIO.bOnCommand AND NOT bLastOnCmd THEN
        tonOnDelay(IN := TRUE, PT := i_tMotionDelay);
        tonOffDelay(IN := FALSE);
    END_IF
    
    // OFF komutu yükselen kenar
    IF io_stIO.bOffCommand AND NOT bLastOffCmd THEN
        tonOffDelay(IN := TRUE, PT := i_tMotionDelay);
        tonOnDelay(IN := FALSE);
    END_IF
    
    // Pozisyon güncelleme
    IF tonOnDelay.Q THEN
        io_stIO.bPositionOn := TRUE;
        io_stIO.bPositionOff := FALSE;
        io_stIO.bPositionTripped := FALSE;
        tonOnDelay(IN := FALSE);
    ELSIF tonOffDelay.Q THEN
        io_stIO.bPositionOn := FALSE;
        io_stIO.bPositionOff := TRUE;
        io_stIO.bPositionTripped := FALSE;
        tonOffDelay(IN := FALSE);
    END_IF
    
    // Hareket halinde
    IF (tonOnDelay.IN OR tonOffDelay.IN) AND NOT tonOnDelay.Q AND NOT tonOffDelay.Q THEN
        io_stIO.bPositionOn := FALSE;
        io_stIO.bPositionOff := FALSE;
        io_stIO.bPositionTripped := FALSE;
    END_IF
END_IF

// Yay durumu simülasyonu
IF i_bSimSpringNotCharged THEN
    io_stIO.bSpringCharged := FALSE;
ELSE
    // OFF konumunda yay otomatik kurulur
    io_stIO.bSpringCharged := io_stIO.bPositionOff OR io_stIO.bPositionOn;
END_IF

// PLC kontrol simülasyonu
io_stIO.bPLCControl := TRUE;

// Önceki komutları sakla
bLastOnCmd := io_stIO.bOnCommand;
bLastOffCmd := io_stIO.bOffCommand;

M_SimulateCircuitBreaker := TRUE;
END_METHOD

METHOD M_SimulateContactor : BOOL
VAR_INPUT
    sContactorName: STRING;         // Kontaktör adı
    i_bSimEnable: BOOL;             // Simülasyon aktif mi?
    i_bSimFeedbackFault: BOOL;      // Geri besleme hatası simülasyonu
    i_bSimWelded: BOOL;             // Yapışma hatası simülasyonu
    i_tFeedbackDelay: TIME;         // Geri besleme gecikmesi
END_VAR
VAR_IN_OUT
    io_stIO: ST_ContactorIO;        // IO structure
END_VAR
VAR_STAT
    tonFeedbackDelay: TON;          // Geri besleme gecikme timer'ı
END_VAR

IF NOT i_bSimEnable THEN
    M_SimulateContactor := FALSE;
    RETURN;
END_IF

// Kontaktör geri besleme simülasyonu
tonFeedbackDelay(IN := io_stIO.bOutput, PT := i_tFeedbackDelay);

IF i_bSimFeedbackFault THEN
    // Geri besleme hatası - feedback gelmiyor
    io_stIO.bFeedback := FALSE;
ELSIF i_bSimWelded THEN
    // Yapışma hatası - feedback sürekli TRUE
    io_stIO.bFeedback := TRUE;
ELSE
    // Normal çalışma
    io_stIO.bFeedback := tonFeedbackDelay.Q;
END_IF

// PLC kontrol simülasyonu (normalde TRUE)
io_stIO.bPLCControl := TRUE;

M_SimulateContactor := TRUE;
END_METHOD

METHOD M_SimulateDisconnector : BOOL
VAR_INPUT
    sDisconnectorName: STRING;              // Ayırıcı adı (örn: 'Disconnector1')
    i_bSimEnable: BOOL;                     // Simülasyon aktif mi?
    i_bSimThermalFault: BOOL;               // Termik hata simülasyonu
    i_bSimEarthSwitchError: BOOL;           // Toprak bıçağı hata simülasyonu
    i_tOnDelay: TIME;                       // ON geçiş süresi
    i_tOffDelay: TIME;                      // OFF geçiş süresi
    i_tContactorDelay: TIME;                // Kontaktör geri bildirim gecikmesi
END_VAR
VAR_IN_OUT
    io_stIO: ST_DisconnectorIO;             // IO structure
END_VAR
VAR_STAT
    tonOnDelay: TON;                        // ON gecikme timer'ı
    tonOffDelay: TON;                       // OFF gecikme timer'ı
    tonContactorDelay: TON;                 // Kontaktör gecikme timer'ı
END_VAR

IF NOT i_bSimEnable THEN
    M_SimulateDisconnector := FALSE;
    RETURN;
END_IF

// ON hareketi simülasyonu
tonOnDelay(IN := io_stIO.bContactorOn_Out, PT := i_tOnDelay);

// OFF hareketi simülasyonu
tonOffDelay(IN := io_stIO.bContactorOff_Out, PT := i_tOffDelay);

// Limit switch simülasyonu
IF tonOnDelay.Q THEN
    io_stIO.bLimitOn := TRUE;
    io_stIO.bLimitOff := FALSE;
ELSIF tonOffDelay.Q THEN
    io_stIO.bLimitOn := FALSE;
    io_stIO.bLimitOff := TRUE;
END_IF

// Ara pozisyon simülasyonu
IF (io_stIO.bContactorOn_Out OR io_stIO.bContactorOff_Out) AND NOT tonOnDelay.Q AND NOT tonOffDelay.Q THEN
    io_stIO.bLimitOn := FALSE;
    io_stIO.bLimitOff := FALSE;
END_IF

// Kontaktör geri bildirim simülasyonu
tonContactorDelay(IN := io_stIO.bContactorOn_Out OR io_stIO.bContactorOff_Out, PT := i_tContactorDelay);

IF tonContactorDelay.Q THEN
    io_stIO.bContactorOn_FB := io_stIO.bContactorOn_Out;
    io_stIO.bContactorOff_FB := io_stIO.bContactorOff_Out;
END_IF

// Toprak bıçağı simülasyonu (ters çalışma)
IF NOT i_bSimEarthSwitchError THEN
    io_stIO.bEarthSwitchOn := io_stIO.bLimitOff;
    io_stIO.bEarthSwitchOff := io_stIO.bLimitOn;
ELSE
    // Hata simülasyonu
    io_stIO.bEarthSwitchOn := FALSE;
    io_stIO.bEarthSwitchOff := FALSE;
END_IF

// Termik hata simülasyonu
io_stIO.bThermalFault := i_bSimThermalFault;

// PLC kontrol simülasyonu (normalde TRUE)
io_stIO.bPLCControl := TRUE;

M_SimulateDisconnector := TRUE;
END_METHOD

END_PROGRAM

// ---- POUs/LVCP1/PRG_LVCP1.TcPOU
PROGRAM PRG_LVCP1
VAR
END_VAR

	PRG_LVCP1_PowerMeasurement();	

	PRG_LVCP1_CompensationCalculate();

	PRG_LVCP1_MainDisconnector();
	
	PRG_Lvcp1_Colors();
	
	PRG_LVCP1_Group1();
	
	PRG_LVCP1_Group2();
	
	PRG_LVCP1_Group3();	
	
	PRG_LVCP1_Group4();	

	PRG_LVCP1_Group5();	

	PRG_LVCP1_Group6();	

	PRG_LVCP1_Group7();	

	PRG_LVCP1_Group8();	

	PRG_LVCP1_Group9();	

	PRG_LVCP1_Group10();

END_PROGRAM

// ---- POUs/LVCP1/PRG_LVCP1_PowerMeasurement.TcPOU
PROGRAM PRG_LVCP1_PowerMeasurement
VAR
	// Enerji Yönetimi
	fbEL3453	: FB_EL3453;	
	stEL3453	: stEL3453;
END_VAR


	fbEL3453(pOut := ADR(stEL3453));

END_PROGRAM

// ---- POUs/EL3453/FB_EL3453.TcPOU
FUNCTION_BLOCK FB_EL3453
VAR_INPUT
	pOut : POINTER TO stEL3453;	
END_VAR
VAR
	EL3453		: MDP5001_341_E4FC35CB;
	
	pSource1 	: UINT := 0;
	AdrCh1	 	: UINT;
	ChNr1		: UINT := 1;
	
	pSource2 	: UINT := 20;
	AdrCh2	 	: UINT;
	ChNr2		: UINT := 2;
	
	pSource3 	: UINT := 25;
	AdrCh3	 	: UINT;
	ChNr3		: UINT := 3;
	
	pSource4 	: UINT := 0;
	AdrCh4	 	: UINT;
	ChNr4		: UINT := 1;
END_VAR



VAR CONSTANT
	sr  : ARRAY[0..32] OF UINT := [2,3,4,5,6,9,11,12,17,21,22,27,28,29,30,33,34,35,36,39,40,41,42,95,98,99,100,165,166,168,169,170,0];
	sr4 : ARRAY[0..34] OF UINT := [15,26,27,28,29,32,33,34,35,38,39,40,41,70,71,72,80,81,82,83,130,131,132,133,136,137,138,139,142,143,144,145,0];
	
	usr : ARRAY[0..18] OF UINT := [3,10,45,46,47,51,52,53,57,58,59,63,64,65,69,75,76,77,0];
	usr4: ARRAY[0..38] OF UINT := [45,46,47,48,49,50,51,52,53,54,55,56,57,58,59,60,61,62,100,101,102,103,104,105,106,107,108,109,110,111,112,113,114,115,116,117,0];
	
END_VAR

EL3453.MDP5001_341_Output.MDP5001_341_Total_Variant_Value_Out_Index_1_REAL := SHL(ChNr1,8) OR AdrCh1;

IF ChNr1 >= 1 AND ChNr1 <= 3 THEN 
	IF AdrCh1 >= 100 AND AdrCh1 < 164  THEN
		AdrCh1 := AdrCh1 + 1;
	ELSIF AdrCh1 >= 170 AND AdrCh1 < 234 THEN
		AdrCh1 := AdrCh1 + 1;
	ELSE
		
		IF sr[pSource1] = 0 THEN
			pSource1 := 0;
			ChNr1 := ChNr1 + 1;
		ELSE
			AdrCh1 := sr[pSource1];
			pSource1 := pSource1 + 1;
		END_IF;
	END_IF		
ELSIF ChNr1 = 4 THEN
	IF sr4[pSource1] = 0 THEN
		pSource1 := 0;
		ChNr1 := 1;
	ELSE
		AdrCh1 := sr4[pSource1];	
		pSource1 := pSource1 + 1;
	END_IF;

END_IF
AddElement( SHR(EL3453.MDP5001_341_Input.MDP5001_341_Total_Variant_Value_In_Index_1_REAL,8), EL3453.MDP5001_341_Input.MDP5001_341_Total_Variant_Value_In_Index_1_REAL AND 16#00FF, EL3453.MDP5001_341_Input.MDP5001_341_Total_Variant_Value_In_Value_1_REAL);
pOut^.Lx[1].fULrms := EL3453.MDP5001_341_Input.MDP5001_341_L1_Basic_Voltage;	
pOut^.Lx[1].fIrms :=EL3453.MDP5001_341_Input.MDP5001_341_L1_Basic_Current;	

pOut^.Lx[1].fPF := EL3453.MDP5001_341_Input.MDP5001_341_L1_Power_Power_Factor;	
pOut^.Lx[1].fP := EL3453.MDP5001_341_Input.MDP5001_341_L1_Power_Active_Power;		
pOut^.Lx[1].fS := EL3453.MDP5001_341_Input.MDP5001_341_L1_Power_Apparent_Power;	
pOut^.Lx[1].fQ := EL3453.MDP5001_341_Input.MDP5001_341_L1_Power_Reactive_Power;	

pOut^.Total.fIerrrmsCalc := EL3453.MDP5001_341_Input.MDP5001_341_Total_Basic_Calculated_Error_Current;	
pOut^.Total.fFreq := EL3453.MDP5001_341_Input.MDP5001_341_Total_Basic_Frequency;							
pOut^.Total.fPF := EL3453.MDP5001_341_Input.MDP5001_341_Total_Basic_Power_Factor;						


//VV2
EL3453.MDP5001_341_Output.MDP5001_341_Total_Variant_Value_Out_Index_2_REAL  := SHL(ChNr2,8) OR AdrCh2;

IF ChNr2 >= 1 AND ChNr2 <= 3 THEN 
	IF AdrCh2 >= 100 AND AdrCh2 < 164  THEN
		AdrCh2 := AdrCh2 + 1;
	ELSIF AdrCh2 >= 170 AND AdrCh2 < 234 THEN
		AdrCh2 := AdrCh2 + 1;
	ELSE
		IF sr[pSource2] = 0 THEN
			pSource2 := 0;
			ChNr2 := ChNr2 + 1;
		ELSE
			AdrCh2 := sr[pSource2];
			pSource2 := pSource2 + 1;
		END_IF;

	END_IF		
ELSIF ChNr2 = 4 THEN
	IF sr4[pSource2] = 0 THEN
		pSource2 := 0;
		ChNr2 := 1;
	ELSE
		AdrCh2 := sr4[pSource2];	
		pSource2 := pSource2 + 1;
	END_IF;

END_IF
 
AddElement( SHR(EL3453.MDP5001_341_Input.MDP5001_341_Total_Variant_Value_In_Index_2_REAL,8), EL3453.MDP5001_341_Input.MDP5001_341_Total_Variant_Value_In_Index_2_REAL AND 16#00FF, EL3453.MDP5001_341_Input.MDP5001_341_Total_Variant_Value_In_Value_2_REAL);
pOut^.Lx[2].fULrms := EL3453.MDP5001_341_Input.MDP5001_341_L2_Basic_Voltage;	
pOut^.Lx[2].fIrms :=EL3453.MDP5001_341_Input.MDP5001_341_L2_Basic_Current;	

pOut^.Lx[2].fPF := EL3453.MDP5001_341_Input.MDP5001_341_L2_Power_Power_Factor;	
pOut^.Lx[2].fP := EL3453.MDP5001_341_Input.MDP5001_341_L2_Power_Active_Power;		
pOut^.Lx[2].fS := EL3453.MDP5001_341_Input.MDP5001_341_L2_Power_Apparent_Power;	
pOut^.Lx[2].fQ := EL3453.MDP5001_341_Input.MDP5001_341_L2_Power_Reactive_Power;	



//VV3
EL3453.MDP5001_341_Output.MDP5001_341_Total_Variant_Value_Out_Index_3_REAL  := SHL(ChNr3,8) OR AdrCh3;
IF ChNr3 >= 1 AND ChNr3 <= 3 THEN 
	IF AdrCh3 >= 100 AND AdrCh3 < 164  THEN
		AdrCh3 := AdrCh3 + 1;
	ELSIF AdrCh3 >= 170 AND AdrCh3 < 234 THEN
		AdrCh3 := AdrCh3 + 1;
	ELSE
		IF sr[pSource3] = 0 THEN
			pSource3 := 0;
			ChNr3 := ChNr3 + 1;
		ELSE
			AdrCh3 := sr[pSource3];
			pSource3 := pSource3 + 1;
		END_IF;

	END_IF		
ELSIF ChNr3 = 4 THEN
	IF sr4[pSource3] = 0 THEN
		pSource3 := 0;
		ChNr3 := 1;
	ELSE
		AdrCh3 := sr4[pSource3];	
		pSource3 := pSource3 + 1;		
	END_IF;

END_IF
 
AddElement( SHR(EL3453.MDP5001_341_Input.MDP5001_341_Total_Variant_Value_In_Index_3_REAL,8), EL3453.MDP5001_341_Input.MDP5001_341_Total_Variant_Value_In_Index_3_REAL AND 16#00FF, EL3453.MDP5001_341_Input.MDP5001_341_Total_Variant_Value_In_Value_3_REAL);
pOut^.Lx[3].fULrms := EL3453.MDP5001_341_Input.MDP5001_341_L3_Basic_Voltage;	
pOut^.Lx[3].fIrms :=EL3453.MDP5001_341_Input.MDP5001_341_L3_Basic_Current;	

pOut^.Lx[3].fPF := EL3453.MDP5001_341_Input.MDP5001_341_L3_Power_Power_Factor;	
pOut^.Lx[3].fP := EL3453.MDP5001_341_Input.MDP5001_341_L3_Power_Active_Power;		
pOut^.Lx[3].fS := EL3453.MDP5001_341_Input.MDP5001_341_L3_Power_Apparent_Power;	
pOut^.Lx[3].fQ := EL3453.MDP5001_341_Input.MDP5001_341_L3_Power_Reactive_Power;	



//VV4
EL3453.MDP5001_341_Output.MDP5001_341_Total_Variant_Value_Out_Index_4_ULINT  := SHL(ChNr4,8) OR AdrCh4;
IF ChNr4 >= 1 AND ChNr4 <= 3 THEN 
	IF usr[pSource4] = 0 THEN
		pSource4 := 0;
		ChNr4 := ChNr4 + 1;
	ELSE
		AdrCh4 := usr[pSource4];
		pSource4 := pSource4 + 1;
	END_IF;

ELSIF ChNr4 = 4 THEN
	IF usr4[pSource4] = 0 THEN
		pSource4 := 0;
		ChNr4 := 1;
	ELSE
		AdrCh4 := usr4[pSource4];	
		pSource4 := pSource4 + 1;
	END_IF;
END_IF
 
AddElementULINT( SHR(EL3453.MDP5001_341_Input.MDP5001_341_Total_Variant_Value_In_Index_4_ULINT,8), EL3453.MDP5001_341_Input.MDP5001_341_Total_Variant_Value_In_Index_4_ULINT AND 16#00FF, EL3453.MDP5001_341_Input.MDP5001_341_Total_Variant_Value_In_Value_4_ULINT);

METHOD AddElement : BOOL
VAR_INPUT
	ChNr : UINT;
	Pos : UINT;
	fElement : REAL;
END_VAR
AddElement := TRUE;

IF ChNr >= 1 AND ChNr <= 3 THEN
	IF Pos >= 100 AND Pos <= 163 THEN
		pOut^.Lx[ChNr].fUL_harm[Pos-100] := fElement;
	ELSIF Pos >= 170 AND Pos <= 233 THEN
		pOut^.Lx[ChNr].fIL_harm[Pos-170] := fElement;
	ELSE	
		CASE Pos OF
			1: pOut^.Lx[ChNr].fULrms 		:= fElement;
			2: pOut^.Lx[ChNr].fUL_peak 		:= fElement;
			
			4: pOut^.Lx[ChNr].fULrms_min 	:= fElement;
			5: pOut^.Lx[ChNr].fULrms_max 	:= fElement;
			//Special Case 6: ULL
			6: 	IF ChNr = 1 THEN
					pOut^.Total.fUL12 		:= fElement;
				ELSIF ChNr = 2 THEN
					pOut^.Total.fUL23		:= fElement;
				ELSE
					pOut^.Total.fUL31		:= fElement;
				END_IF
			
			
			8: pOut^.Lx[ChNr].fIrms 		:= fElement;
			9: pOut^.Lx[ChNr].fI_peak 		:= fElement;
			
			11: pOut^.Lx[ChNr].fIrms_min 	:= fElement;
			12: pOut^.Lx[ChNr].fIrms_max 	:= fElement;
			
			17: pOut^.Lx[ChNr].fFreq 		:= fElement;
			
			21: pOut^.Lx[ChNr].fPhi		 	:= fElement;
			22: pOut^.Lx[ChNr].fCosPhi	 	:= fElement;
			23: pOut^.Lx[ChNr].fPF		 	:= fElement;
			
			26: pOut^.Lx[ChNr].fP 			:= fElement;
			27: pOut^.Lx[ChNr].fP_avg 		:= fElement;
			28: pOut^.Lx[ChNr].fP_min 		:= fElement;
			29: pOut^.Lx[ChNr].fP_max 		:= fElement;
			30: pOut^.Lx[ChNr].fP_fund 		:= fElement;
						
			32: pOut^.Lx[ChNr].fS 			:= fElement;
			33: pOut^.Lx[ChNr].fS_avg 		:= fElement;
			34: pOut^.Lx[ChNr].fS_min 		:= fElement;
			35: pOut^.Lx[ChNr].fS_max 		:= fElement;
			36: pOut^.Lx[ChNr].fS_fund 		:= fElement;
						
			38: pOut^.Lx[ChNr].fQ 			:= fElement;
			39: pOut^.Lx[ChNr].fQ_avg 		:= fElement;
			40: pOut^.Lx[ChNr].fQ_min 		:= fElement;
			41: pOut^.Lx[ChNr].fQ_max 		:= fElement;
			42: pOut^.Lx[ChNr].fQ_fund 		:= fElement;
			
			95: pOut^.Lx[ChNr].fUL_THD	 	:= fElement;
			98: pOut^.Lx[ChNr].fULrms_fund 	:= fElement;
			99: pOut^.Lx[ChNr].fUL_harmrf 	:= fElement;
			
			165: pOut^.Lx[ChNr].fI_THD 		:= fElement;
			166: pOut^.Lx[ChNr].fI_TDD 		:= fElement;
			168: pOut^.Lx[ChNr].fIrms_fund	:= fElement;
			169: pOut^.Lx[ChNr].fIL_harmrf	:= fElement;
			
			ELSE 
				AddElement := FALSE;
		END_CASE
	END_IF
ELSIF ChNr = 4 THEN
	CASE Pos OF
		8:  pOut^.Total.fIerrrmsCalc	:= fElement;
		15: pOut^.Total.fInrms	 		:= fElement;
		17: pOut^.Total.fFreq			:= fElement;
		23: pOut^.Total.fPF		 		:= fElement;
		
		26: pOut^.Total.fP		 		:= fElement;
		27: pOut^.Total.fP_avg	 		:= fElement; 
		28: pOut^.Total.fP_min	 		:= fElement;
		29: pOut^.Total.fP_max	 		:= fElement;
		
		32: pOut^.Total.fS		 		:= fElement;
		33: pOut^.Total.fS_avg	 		:= fElement; 
		34: pOut^.Total.fS_min	 		:= fElement;
		35: pOut^.Total.fS_max	 		:= fElement;
		
		38: pOut^.Total.fQtot		 	:= fElement;
		39: pOut^.Total.fQtot_avg	 	:= fElement; 
		40: pOut^.Total.fQtot_min	 	:= fElement;
		41: pOut^.Total.fQtot_max	 	:= fElement;
		
		70: pOut^.Total.fPhiL1L2	 	:= fElement;
		71: pOut^.Total.fPhiL1L3	 	:= fElement;
		72: pOut^.Total.fUnbalance		:= fElement;
		
		80: pOut^.Total.fPQF		 	:= fElement;
		81: pOut^.Total.fPQF_avg	 	:= fElement;
		82: pOut^.Total.fPQF_min	 	:= fElement;
		83: pOut^.Total.fPQF_max	 	:= fElement;
		
		130: pOut^.Total.fP_fund		:= fElement;
		131: pOut^.Total.fP_fund_avg	:= fElement;
		132: pOut^.Total.fP_fund_min	:= fElement;
		133: pOut^.Total.fP_fund_max	:= fElement;

		136: pOut^.Total.fS_fund		:= fElement;
		137: pOut^.Total.fS_fund_avg	:= fElement;
		138: pOut^.Total.fS_fund_min	:= fElement;
		139: pOut^.Total.fS_fund_max	:= fElement;
		
		142: pOut^.Total.fQ_fund		:= fElement;
		143: pOut^.Total.fQ_fund_avg	:= fElement;
		144: pOut^.Total.fQ_fund_min	:= fElement;
		145: pOut^.Total.fQ_fund_max	:= fElement;
		
		ELSE 
			AddElement := FALSE;
		END_CASE
ELSE
	AddElement := FALSE;
END_IF
END_METHOD

METHOD AddElementULINT : BOOL
VAR_INPUT
	ChNr : UINT;
	Pos : UINT;
	uElement : ULINT;
END_VAR
AddElementULINT := TRUE;

IF ChNr >= 1 AND ChNr <= 3 THEN
	CASE Pos OF
		3 :	pOut^.Lx[ChNr].ulUL_ZC 			:= uElement;
		10:	pOut^.Lx[ChNr].ulI_ZC 			:= uElement;
		
		45: pOut^.Lx[ChNr].lEP	 			:= uElement;
		46: pOut^.Lx[ChNr].ulEP_pos	 		:= uElement;
		47: pOut^.Lx[ChNr].ulEP_neg	 		:= uElement;
		
		51: pOut^.Lx[ChNr].lES	 			:= uElement;
		52: pOut^.Lx[ChNr].ulES_pos	 		:= uElement;
		53: pOut^.Lx[ChNr].ulES_neg	 		:= uElement;
		
		57: pOut^.Lx[ChNr].lEQ	 			:= uElement;
		58: pOut^.Lx[ChNr].ulEQ_pos			:= uElement;
		59: pOut^.Lx[ChNr].ulEQ_neg			:= uElement;
		
		63: pOut^.Lx[ChNr].lEP_fund	 		:= uElement;
		64: pOut^.Lx[ChNr].ulEP_fund_pos 	:= uElement;
		65: pOut^.Lx[ChNr].ulEP_fund_neg 	:= uElement;
		
		69: pOut^.Lx[ChNr].lES_fund	 		:= uElement;
		70: pOut^.Lx[ChNr].ulES_fund_pos 	:= uElement;
		71: pOut^.Lx[ChNr].ulES_fund_neg 	:= uElement;
		
		75: pOut^.Lx[ChNr].lEQ_fund	 		:= uElement;
		76: pOut^.Lx[ChNr].ulEQ_fund_pos	:= uElement;
		77: pOut^.Lx[ChNr].ulEQ_fund_neg	:= uElement;
		
		
		ELSE 
			AddElementULINT := FALSE;
	END_CASE
ELSIF ChNr = 4 THEN
	CASE Pos OF
		
		45 : pOut^.Total.lEP				:= uElement;
		46 : pOut^.Total.ulEP_pos			:= uElement;
		47 : pOut^.Total.ulEP_neg	 		:= uElement;
		
		48 : pOut^.Total.lEP_int 			:= uElement;
		49 : pOut^.Total.ulEP_int_pos		:= uElement;
		50 : pOut^.Total.ulEP_int_neg		:= uElement;
		
		51 : pOut^.Total.lES	 			:= uElement;
		52 : pOut^.Total.ulES_pos			:= uElement;
		53 : pOut^.Total.ulES_neg			:= uElement;
		
		54 : pOut^.Total.lES_int	 		:= uElement;
		55 : pOut^.Total.ulES_int_pos		:= uElement;
		56 : pOut^.Total.ulES_int_neg		:= uElement;

		57 : pOut^.Total.lEQ	 			:= uElement;
		58 : pOut^.Total.ulEQ_pos			:= uElement;
		59 : pOut^.Total.ulEQ_neg			:= uElement;		
		
		60 : pOut^.Total.lEQ_int	 		:= uElement;
		61 : pOut^.Total.ulEQ_int_pos		:= uElement;
		62 : pOut^.Total.ulEQ_int_neg		:= uElement;
										
		100: pOut^.Total.lEP_fund	 		:= uElement;
		101: pOut^.Total.ulEP_fund_pos		:= uElement;
		102: pOut^.Total.ulEP_fund_neg	 	:= uElement;
		
		103: pOut^.Total.lEP_fund_int 		:= uElement;
		104: pOut^.Total.ulEP_fund_int_pos	:= uElement;
		105: pOut^.Total.ulEP_fund_int_neg	:= uElement;
		
		106: pOut^.Total.lES_fund	 		:= uElement;
		107: pOut^.Total.ulES_fund_pos		:= uElement;
		108: pOut^.Total.ulES_fund_neg		:= uElement;
		
		109: pOut^.Total.lES_fund_int	 	:= uElement;
		110: pOut^.Total.ulES_fund_int_pos	:= uElement;
		111: pOut^.Total.ulES_fund_int_neg	:= uElement;

		112: pOut^.Total.lEQ_fund	 		:= uElement;
		113: pOut^.Total.ulEQ_fund_pos		:= uElement;
		114: pOut^.Total.ulEQ_fund_neg		:= uElement;		
		
		115: pOut^.Total.lEQ_fund_int	 	:= uElement;
		116: pOut^.Total.ulEQ_fund_int_pos	:= uElement;
		117: pOut^.Total.ulEQ_fund_int_neg	:= uElement;
		
		ELSE 
				AddElementULINT := FALSE;
		END_CASE
ELSE
	AddElementULINT := FALSE;
END_IF
END_METHOD

END_FUNCTION_BLOCK

// ---- POUs/LVCP1/PRG_LVCP1_CompensationCalculate.TcPOU
PROGRAM PRG_LVCP1_CompensationCalculate
VAR
    fbCompensationCalc : FB_CompensationCalculator;
    bCalculate : BOOL := TRUE;              // Sürekli hesaplama için
    nActiveGroups : INT := 10;              // Toplam 10 grup
    
    // Outputs
    stHMIData : ST_CompensationHMI;
    asCapacitorTags : ARRAY[0..99] OF STRING(30);
    nActiveTags : INT;
    
    // Özet bilgiler
    rTotalPower : REAL;
    nTotalCapacitors : INT;
    nActiveGroupCount : INT;
END_VAR

// Grup sayısını güncelle
GVL_LVCP1.nConfiguredGroups := nActiveGroups;

// Hesaplama
fbCompensationCalc(
    bExecute 				:= bCalculate,
    bGroupActive 			:= GVL_LVCP1.abGroupActive,
    stGroupConfig 			:= GVL_LVCP1.astCompensationGroups,
    nActiveGroups 			:= GVL_LVCP1.nConfiguredGroups,
    stHMI 					=> stHMIData,
    asActiveCapacitorTags 	=> asCapacitorTags,
    nActiveCapacitorCount 	=> nActiveTags
);

// Özet bilgiler
rTotalPower 		:= stHMIData.stSummary.rTotalActivePower;
nTotalCapacitors 	:= stHMIData.stSummary.nTotalActiveCapacitors;
nActiveGroupCount 	:= stHMIData.stSummary.nActiveGroupCount;

END_PROGRAM

// ---- _ES/14_CompensationGroup/FB_CompensationCalculator.TcPOU
FUNCTION_BLOCK FB_CompensationCalculator

VAR_INPUT
    bExecute : BOOL;                                                                            // Hesaplama tetikleme
    bGroupActive : ARRAY[0..GVL_CompensationGroup.MAX_COMPENSATION_GROUPS-1] OF BOOL;          // Grup aktif durumları
    stGroupConfig : ARRAY[0..GVL_CompensationGroup.MAX_COMPENSATION_GROUPS-1] OF ST_CompensationGroup;  // Grup konfigürasyonları
    nActiveGroups : INT;                                                                        // Kullanımdaki grup sayısı
END_VAR

VAR_OUTPUT
    stHMI : ST_CompensationHMI;                                                                // HMI için tüm bilgiler
    asActiveCapacitorTags : ARRAY[0..GVL_CompensationGroup.MAX_TOTAL_CAPACITORS-1] OF STRING(GVL_CompensationGroup.MAX_TAG_LENGTH); // Aktif kondansatör etiketleri
    nActiveCapacitorCount : INT;                                                                // asActiveCapacitorTags dizisindeki geçerli eleman sayısı
END_VAR

VAR
    i : INT;                                                                                    // Döngü değişkeni
    j : INT;                                                                                    // İç döngü değişkeni
    nTagIndex : INT;                                                                            // Etiket dizisi indeksi
    bExecuteOld : BOOL;                                                                         // Execute rising edge detection
    bInitialized : BOOL;                                                                        // İlk çalışma kontrolü
END_VAR

// İlk çalışmada veya Execute rising edge'de init ve kontrol yap
IF NOT bInitialized OR (bExecute AND NOT bExecuteOld) THEN
    // Initialization
    M_Init();
    
    // Hata kontrolü
    IF NOT M_CheckErrors() THEN
        bInitialized := TRUE;
        bExecuteOld := bExecute;
        RETURN;
    END_IF
    
    // Config bilgilerini kopyala
    stHMI.stConfig.nConfiguredGroups := nActiveGroups;
    FOR i := 0 TO nActiveGroups - 1 DO
        stHMI.stConfig.astGroupConfig[i] := stGroupConfig[i];
    END_FOR
    
    bInitialized := TRUE;
END_IF

// Her çevrimde sadece hesaplama yap
IF bInitialized AND NOT stHMI.stDiagnostic.bError THEN
    M_Calculate();
END_IF

bExecuteOld := bExecute;

METHOD M_Calculate : BOOL
VAR
    i : INT;
    j : INT;
    rGroupTotalPower : REAL;
END_VAR

// Her grubu kontrol et ve hesapla
FOR i := 0 TO nActiveGroups - 1 DO
    // Grup aktif mi?
    IF bGroupActive[i] THEN
        // Bu gruptaki kondansatör sayısını toplama ekle
        stHMI.stSummary.nTotalActiveCapacitors := stHMI.stSummary.nTotalActiveCapacitors + stGroupConfig[i].nQuantity;
        
        // Bu grubun toplam gücünü hesapla
        rGroupTotalPower := stGroupConfig[i].rPower * stGroupConfig[i].nQuantity;
        stHMI.stGroupDetails.arGroupPower[i] := rGroupTotalPower;
        stHMI.stSummary.rTotalActivePower := stHMI.stSummary.rTotalActivePower + rGroupTotalPower;
        
        // Grup detaylarını güncelle
        stHMI.stGroupDetails.abGroupActive[i] := TRUE;
        stHMI.stGroupDetails.anGroupCapacitorCount[i] := stGroupConfig[i].nQuantity;
        stHMI.stSummary.nActiveGroupCount := stHMI.stSummary.nActiveGroupCount + 1;
        
        // Etiketleri oluştur
        FOR j := 1 TO stGroupConfig[i].nQuantity DO
            IF nTagIndex < GVL_CompensationGroup.MAX_TOTAL_CAPACITORS THEN
                asActiveCapacitorTags[nTagIndex] := CONCAT(stGroupConfig[i].sTagPrefix, CONCAT('_', INT_TO_STRING(j)));
                nTagIndex := nTagIndex + 1;
            END_IF
        END_FOR
    END_IF
END_FOR

nActiveCapacitorCount := nTagIndex;
M_Calculate := TRUE;
END_METHOD

METHOD M_CheckErrors : BOOL
VAR
    i : INT;
    bErrorFound : BOOL := FALSE;
END_VAR

// Input kontrolü - grup sayısı
IF nActiveGroups < 0 OR nActiveGroups > GVL_CompensationGroup.MAX_COMPENSATION_GROUPS THEN
    stHMI.stDiagnostic.bError := TRUE;
    stHMI.stDiagnostic.eError := E_CompensationError.ERROR_INVALID_GROUP_COUNT;
    stHMI.stDiagnostic.wsErrorMessage := "Geçersiz grup sayısı";
    M_CheckErrors := FALSE;
    RETURN;
END_IF

// Her grup için config kontrolü
FOR i := 0 TO nActiveGroups - 1 DO
    // Negatif kondansatör sayısı kontrolü
    IF stGroupConfig[i].nQuantity < 0 THEN
        stHMI.stDiagnostic.bError := TRUE;
        stHMI.stDiagnostic.eError := E_CompensationError.ERROR_NEGATIVE_QUANTITY;
        stHMI.stDiagnostic.wsErrorMessage := WCONCAT("Grup ", WCONCAT(INT_TO_WSTRING(i+1), " için negatif kondansatör sayısı"));
        M_CheckErrors := FALSE;
        RETURN;
    END_IF
    
    // Negatif güç kontrolü
    IF stGroupConfig[i].rPower < 0 THEN
        stHMI.stDiagnostic.bError := TRUE;
        stHMI.stDiagnostic.eError := E_CompensationError.ERROR_NEGATIVE_POWER;
        stHMI.stDiagnostic.wsErrorMessage := WCONCAT("Grup ", WCONCAT(INT_TO_WSTRING(i+1), " için negatif güç değeri"));
        M_CheckErrors := FALSE;
        RETURN;
    END_IF
END_FOR

// Maksimum kondansatör sayısı kontrolü (hesaplama sonrası kontrol için)
IF stHMI.stSummary.nTotalActiveCapacitors > GVL_CompensationGroup.MAX_TOTAL_CAPACITORS THEN
    stHMI.stDiagnostic.bError := TRUE;
    stHMI.stDiagnostic.eError := E_CompensationError.ERROR_MAX_CAPACITOR_EXCEEDED;
    stHMI.stDiagnostic.wsErrorMessage := WCONCAT("Maksimum kondansatör sayısı aşıldı: ", INT_TO_WSTRING(stHMI.stSummary.nTotalActiveCapacitors));
    M_CheckErrors := FALSE;
    RETURN;
END_IF

// Hata yok
M_CheckErrors := TRUE;
END_METHOD

METHOD M_Init : BOOL
VAR
    i : INT;
END_VAR
// Başlangıç değerlerini sıfırla
stHMI.stSummary.nTotalActiveCapacitors := 0;
stHMI.stSummary.rTotalActivePower := 0;
stHMI.stSummary.nActiveGroupCount := 0;

stHMI.stDiagnostic.bError := FALSE;
stHMI.stDiagnostic.eError := E_CompensationError.ERROR_NONE;
stHMI.stDiagnostic.wsErrorMessage := "";

nTagIndex := 0;
nActiveCapacitorCount := 0;

// Grup detaylarını sıfırla
FOR i := 0 TO GVL_CompensationGroup.MAX_COMPENSATION_GROUPS - 1 DO
    stHMI.stGroupDetails.abGroupActive[i] := FALSE;
    stHMI.stGroupDetails.arGroupPower[i] := 0;
    stHMI.stGroupDetails.anGroupCapacitorCount[i] := 0;
END_FOR

// Etiket dizisini temizle
FOR i := 0 TO GVL_CompensationGroup.MAX_TOTAL_CAPACITORS - 1 DO
    asActiveCapacitorTags[i] := '';
END_FOR

M_Init := TRUE;
END_METHOD

END_FUNCTION_BLOCK

// ---- POUs/LVCP1/PRG_LVCP1_MainDisconnector.TcPOU
PROGRAM PRG_LVCP1_MainDisconnector
VAR
    // Function Block Instance
    fbDisconnector		: FB_DisconnectorControl;
	
	stDisconnectorIO	: ST_DisconnectorIO;
	
    
    // Başlangıç konfigürasyonu için flag
    bInitDone: BOOL := FALSE;	
END_VAR

IF NOT bInitDone THEN
	bInitDone := TRUE;
	RETURN;
END_IF

//*************************************************************************
// Ana Besleme Ayırıcısı
// +EP6-8CB1
//*************************************************************************
fbDisconnector(
    // Fiziksel Girişler
    bContactorOn_FB 	:= stDisconnectorIO.bContactorOn_FB,
    bContactorOff_FB 	:= stDisconnectorIO.bContactorOff_FB,
    bLimitOn 			:= stDisconnectorIO.bLimitOn,
    bLimitOff 			:= stDisconnectorIO.bLimitOff,
    bThermalFault 		:= stDisconnectorIO.bThermalFault,
    bEarthSwitchOn 		:= stDisconnectorIO.bEarthSwitchOn,
    bEarthSwitchOff 	:= stDisconnectorIO.bEarthSwitchOff,
    bPLCControl 		:= stDisconnectorIO.bPLCControl,
    
    // Güvenlik Girişleri
    bSafetyLoop 		:= GVL_Alarm.bSafetyLoop,
    bInterlock 			:= FALSE,
    
    // Sistem Girişleri
    bMasterReset 		:= GVL_Alarm.bMasterReset,
    
    // HMI Bağlantısı
    stHMI 				:= GVL_LVCP1.stMainDisconnectorHMI,
    
    // Fiziksel Çıkışlar
    bContactorOn_Out 	=> stDisconnectorIO.bContactorOn_Out,
    bContactorOff_Out 	=> stDisconnectorIO.bContactorOff_Out
);

METHOD M_Init : BOOL
VAR_INPUT
END_VAR

GVL_LVCP1.stMainDisconnectorHMI.stConfig.bEarthSwitchExists := TRUE;
GVL_LVCP1.stMainDisconnectorHMI.stConfig.bGrounded := TRUE;
GVL_LVCP1.stMainDisconnectorHMI.stConfig.bInterlockEnable := TRUE;
GVL_LVCP1.stMainDisconnectorHMI.stConfig.dwOperationLimit := 10000;
GVL_LVCP1.stMainDisconnectorHMI.stConfig.nPhaseCount := 3;
GVL_LVCP1.stMainDisconnectorHMI.stConfig.rRatedCurrent := 1600.0;
GVL_LVCP1.stMainDisconnectorHMI.stConfig.rRatedVoltage := 1000.0;
GVL_LVCP1.stMainDisconnectorHMI.stConfig.sProductCode := '';
GVL_LVCP1.stMainDisconnectorHMI.stConfig.sProjectCode := '+EP6-8CB1';
GVL_LVCP1.stMainDisconnectorHMI.stConfig.tContactorDelay := T#500MS;
GVL_LVCP1.stMainDisconnectorHMI.stConfig.tMotionTimeout := T#50S;
END_METHOD

END_PROGRAM

// ---- POUs/LVCP1/PRG_LVCP1_Colors.TcPOU
PROGRAM PRG_LVCP1_Colors
VAR
	arrLine : ARRAY[1..4] OF E_LineColors;
	arrCapacitorSchemaColor : ARRAY[1..10] OF ST_CapacitorSchemaColorWithContactor;

	i : INT;
	bInitDone : BOOL;
END_VAR

IF NOT bInitDone THEN
	ACT_ContactorConfigurations();
	bInitDone := TRUE;
END_IF

//line1
arrLine[1] := E_LineColors.Energised_Red;

//line2
arrLine[2] := arrLine[1];

//line3
arrLine[3] := arrLine[2];

//line4
arrLine[4] := arrLine[3];

//şemaları kendi içerisinde kontrol edicez
FOR i:=1 TO 10 DO
	arrCapacitorSchemaColor[i].GroundColor := E_LineColors.Grounded_Green;
	arrCapacitorSchemaColor[i].BottomLineColor2 := E_LineColors.Grounded_Green;

	//topline
	arrCapacitorSchemaColor[i].TopLineColor := arrLine[4];
	
	//bottomLine - şema üzerinde ayırıcının altındaki her iki line birbiri ile bağlantılı olduğu için tek yerden yönetiliyor
	IF arrCapacitorSchemaColor[i].ContactorPosition = E_ContactorPosition.ON THEN
		arrCapacitorSchemaColor[i].BottomLineColor := arrCapacitorSchemaColor[i].TopLineColor;
	ELSE
		arrCapacitorSchemaColor[i].BottomLineColor := E_LineColors.Default;
	END_IF
	
	//capacitor
	arrCapacitorSchemaColor[i].CapacitorColor := arrCapacitorSchemaColor[i].BottomLineColor;
	
END_FOR

ACTION ACT_ContactorConfigurations:
arrCapacitorSchemaColor[1].ContactorPosition := GVL_LVCP1.stGroup1_ContactorHMI.stStatus.ePosition;
arrCapacitorSchemaColor[2].ContactorPosition := GVL_LVCP1.stGroup2_ContactorHMI.stStatus.ePosition;
arrCapacitorSchemaColor[3].ContactorPosition := GVL_LVCP1.stGroup3_ContactorHMI.stStatus.ePosition;
arrCapacitorSchemaColor[4].ContactorPosition := GVL_LVCP1.stGroup4_ContactorHMI.stStatus.ePosition;
arrCapacitorSchemaColor[5].ContactorPosition := GVL_LVCP1.stGroup5_ContactorHMI.stStatus.ePosition;
arrCapacitorSchemaColor[6].ContactorPosition := GVL_LVCP1.stGroup6_ContactorHMI.stStatus.ePosition;
arrCapacitorSchemaColor[7].ContactorPosition := GVL_LVCP1.stGroup7_ContactorHMI.stStatus.ePosition;
arrCapacitorSchemaColor[8].ContactorPosition := GVL_LVCP1.stGroup8_ContactorHMI.stStatus.ePosition;
arrCapacitorSchemaColor[9].ContactorPosition := GVL_LVCP1.stGroup9_ContactorHMI.stStatus.ePosition;
arrCapacitorSchemaColor[10].ContactorPosition := GVL_LVCP1.stGroup10_ContactorHMI.stStatus.ePosition;
END_ACTION

END_PROGRAM

// ---- POUs/LVCP1/PRG_LVCP1_Group1.TcPOU
PROGRAM PRG_LVCP1_Group1
VAR
    // Function Block Instance
    fbContactor: FB_ContactorControl;

    // Contactor 1 IO Structure  
    stContactor_IO: ST_ContactorIO;
    
    // Başlangıç konfigürasyonu için flag
    bContactorInitDone: BOOL := FALSE;
    bCapacitorInitDone: BOOL := FALSE;	
END_VAR



	M_Contactor();
	
	M_Capacitor();

METHOD M_Capacitor : BOOL
VAR
    nGroupIndex : INT;
END_VAR
	nGroupIndex := 0;  // Grup 1 için index
	
	IF NOT bCapacitorInitDone THEN
	
		// Grup 1 değerlerini ata
		GVL_LVCP1.astCompensationGroups[nGroupIndex].rPower := 25.0;
		GVL_LVCP1.astCompensationGroups[nGroupIndex].rVoltage := 450.0;
		GVL_LVCP1.astCompensationGroups[nGroupIndex].nQuantity := 10;
		GVL_LVCP1.astCompensationGroups[nGroupIndex].sTagPrefix := '+EP6-16C1';
		GVL_LVCP1.astCompensationGroups[nGroupIndex].sProductCode := 'ENT.CXD-450-25';
		
		bCapacitorInitDone := TRUE;
	END_IF
	
	// Grup 1 aktif durumu
	GVL_LVCP1.abGroupActive[nGroupIndex] := stContactor_IO.bFeedback;
	
	M_Capacitor := TRUE;
END_METHOD

METHOD M_Contactor : BOOL
VAR_INPUT
END_VAR
IF NOT bContactorInitDone THEN
    // Konfigürasyon parametreleri
    GVL_LVCP1.stGroup1_ContactorHMI.stConfig.sProjectCode := '+EP6-17K1';
    GVL_LVCP1.stGroup1_ContactorHMI.stConfig.sProductCode := 'SCH LC1G630LSEA';
    GVL_LVCP1.stGroup1_ContactorHMI.stConfig.rRatedCurrent := 630.0;
    GVL_LVCP1.stGroup1_ContactorHMI.stConfig.rRatedVoltage := 1000.0;
    GVL_LVCP1.stGroup1_ContactorHMI.stConfig.nPhaseCount := 3;
    GVL_LVCP1.stGroup1_ContactorHMI.stConfig.tFeedbackDelay := T#500MS;
    GVL_LVCP1.stGroup1_ContactorHMI.stConfig.tWeldedDelay := T#2S;
    GVL_LVCP1.stGroup1_ContactorHMI.stConfig.dwOperationLimit := 100000;
    // Başlangıç bakım sayacı
    GVL_LVCP1.stGroup1_ContactorHMI.stStatistics.dwRemainingOperations := GVL_LVCP1.stGroup1_ContactorHMI.stConfig.dwOperationLimit;
	
	bContactorInitDone := TRUE;
END_IF	
	
// Function Block Çağrısı
fbContactor(
    // Fiziksel Girişler
    bFeedback 		:= stContactor_IO.bFeedback,
    bPLCControl 	:= stContactor_IO.bPLCControl,
    
    // Güvenlik Girişleri
    bSafetyLoop 	:= GVL_Alarm.bSafetyLoop,
    bInterlock 		:= FALSE,
    
    // Sistem Girişleri
    bMasterReset 	:= GVL_Alarm.bMasterReset,
    
    // HMI Bağlantısı
    stHMI 			:= GVL_LVCP1.stGroup1_ContactorHMI,
    
    // Fiziksel Çıkış
    bOutput 		=> stContactor_IO.bOutput
);

// SQL Kayıt İşlemi
IF GVL_LVCP1.stGroup1_ContactorHMI.stStatistics.bNewOperationFlag THEN
    // SQL kayıt fonksiyonunu çağır
    GVL_LVCP1.stGroup1_ContactorHMI.stStatistics.bNewOperationFlag := FALSE;
END_IF
END_METHOD

END_PROGRAM

// ---- POUs/LVCP1/PRG_LVCP1_Group2.TcPOU
PROGRAM PRG_LVCP1_Group2
VAR
    // Function Block Instance
    fbContactor: FB_ContactorControl;

    // Contactor 1 IO Structure  
    stContactor_IO: ST_ContactorIO;
    
    // Başlangıç konfigürasyonu için flag
    bContactorInitDone: BOOL := FALSE;
    bCapacitorInitDone: BOOL := FALSE;	
END_VAR



	M_Contactor();
	
	M_Capacitor();

METHOD M_Capacitor : BOOL
VAR
    nGroupIndex : INT;
END_VAR

nGroupIndex := 1;  // Grup 2 için index

IF NOT bCapacitorInitDone THEN
    // Grup 2 değerlerini ata
    GVL_LVCP1.astCompensationGroups[nGroupIndex].rPower := 25.0;
    GVL_LVCP1.astCompensationGroups[nGroupIndex].rVoltage := 450.0;
    GVL_LVCP1.astCompensationGroups[nGroupIndex].nQuantity := 8;
    GVL_LVCP1.astCompensationGroups[nGroupIndex].sTagPrefix := '+EP6-19C1';
    GVL_LVCP1.astCompensationGroups[nGroupIndex].sProductCode := 'ENT.CXD-450-25';
    
    bCapacitorInitDone := TRUE;
END_IF

// Grup 2 aktif durumu
GVL_LVCP1.abGroupActive[nGroupIndex] := stContactor_IO.bFeedback;

M_Capacitor := TRUE;
END_METHOD

METHOD M_Contactor : BOOL
VAR_INPUT
END_VAR

IF NOT bContactorInitDone THEN
    // Konfigürasyon parametreleri
    GVL_LVCP1.stGroup2_ContactorHMI.stConfig.sProjectCode := '+EP6-20K1';
    GVL_LVCP1.stGroup2_ContactorHMI.stConfig.sProductCode := 'SCH LC1G500LSEA';
    GVL_LVCP1.stGroup2_ContactorHMI.stConfig.rRatedCurrent := 500.0;
    GVL_LVCP1.stGroup2_ContactorHMI.stConfig.rRatedVoltage := 1000.0;
    GVL_LVCP1.stGroup2_ContactorHMI.stConfig.nPhaseCount := 3;
    GVL_LVCP1.stGroup2_ContactorHMI.stConfig.tFeedbackDelay := T#500MS;
    GVL_LVCP1.stGroup2_ContactorHMI.stConfig.tWeldedDelay := T#2S;
    GVL_LVCP1.stGroup2_ContactorHMI.stConfig.dwOperationLimit := 100000;
    
    // Başlangıç bakım sayacı
    GVL_LVCP1.stGroup2_ContactorHMI.stStatistics.dwRemainingOperations := GVL_LVCP1.stGroup2_ContactorHMI.stConfig.dwOperationLimit;
    
    bContactorInitDone := TRUE;
END_IF

// Function Block Çağrısı
fbContactor(
    // Fiziksel Girişler
    bFeedback := stContactor_IO.bFeedback,
    bPLCControl := stContactor_IO.bPLCControl,
    
    // Güvenlik Girişleri
    bSafetyLoop := GVL_Alarm.bSafetyLoop,
    bInterlock := FALSE,
    
    // Sistem Girişleri
    bMasterReset := GVL_Alarm.bMasterReset,
    
    // HMI Bağlantısı
    stHMI := GVL_LVCP1.stGroup2_ContactorHMI,
    
    // Fiziksel Çıkış
    bOutput => stContactor_IO.bOutput
);

M_Contactor := TRUE;
END_METHOD

END_PROGRAM

// ---- POUs/LVCP1/PRG_LVCP1_Group3.TcPOU
PROGRAM PRG_LVCP1_Group3
VAR
    // Function Block Instance
    fbContactor: FB_ContactorControl;

    // Contactor 1 IO Structure  
    stContactor_IO: ST_ContactorIO;
    
    // Başlangıç konfigürasyonu için flag
    bContactorInitDone: BOOL := FALSE;
    bCapacitorInitDone: BOOL := FALSE;	
END_VAR



	M_Contactor();
	
	M_Capacitor();

METHOD M_Capacitor : BOOL
VAR
    nGroupIndex : INT;
END_VAR

nGroupIndex := 2;  // Grup 3 için index

IF NOT bCapacitorInitDone THEN
    // Grup 3 değerlerini ata
    GVL_LVCP1.astCompensationGroups[nGroupIndex].rPower := 25.0;
    GVL_LVCP1.astCompensationGroups[nGroupIndex].rVoltage := 450.0;
    GVL_LVCP1.astCompensationGroups[nGroupIndex].nQuantity := 6;
    GVL_LVCP1.astCompensationGroups[nGroupIndex].sTagPrefix := '+EP6-22C1';
    GVL_LVCP1.astCompensationGroups[nGroupIndex].sProductCode := 'ENT.CXD-450-25';
    
    bCapacitorInitDone := TRUE;
END_IF

// Grup 3 aktif durumu
GVL_LVCP1.abGroupActive[nGroupIndex] := stContactor_IO.bFeedback;

M_Capacitor := TRUE;
END_METHOD

METHOD M_Contactor : BOOL
VAR_INPUT
END_VAR
IF NOT bContactorInitDone THEN
    // Konfigürasyon parametreleri
    GVL_LVCP1.stGroup3_ContactorHMI.stConfig.sProjectCode := '+EP6-23K1';
    GVL_LVCP1.stGroup3_ContactorHMI.stConfig.sProductCode := 'SCH LC1G500LSEA';
    GVL_LVCP1.stGroup3_ContactorHMI.stConfig.rRatedCurrent := 500.0;
    GVL_LVCP1.stGroup3_ContactorHMI.stConfig.rRatedVoltage := 1000.0;
    GVL_LVCP1.stGroup3_ContactorHMI.stConfig.nPhaseCount := 3;
    GVL_LVCP1.stGroup3_ContactorHMI.stConfig.tFeedbackDelay := T#500MS;
    GVL_LVCP1.stGroup3_ContactorHMI.stConfig.tWeldedDelay := T#2S;
    GVL_LVCP1.stGroup3_ContactorHMI.stConfig.dwOperationLimit := 100000;
    
    // Başlangıç bakım sayacı
    GVL_LVCP1.stGroup3_ContactorHMI.stStatistics.dwRemainingOperations := GVL_LVCP1.stGroup3_ContactorHMI.stConfig.dwOperationLimit;
    
    bContactorInitDone := TRUE;
END_IF

// Function Block Çağrısı
fbContactor(
    // Fiziksel Girişler
    bFeedback := stContactor_IO.bFeedback,
    bPLCControl := stContactor_IO.bPLCControl,
    
    // Güvenlik Girişleri
    bSafetyLoop := GVL_Alarm.bSafetyLoop,
    bInterlock := FALSE,
    
    // Sistem Girişleri
    bMasterReset := GVL_Alarm.bMasterReset,
    
    // HMI Bağlantısı
    stHMI := GVL_LVCP1.stGroup3_ContactorHMI,
    
    // Fiziksel Çıkış
    bOutput => stContactor_IO.bOutput
);

M_Contactor := TRUE;
END_METHOD

END_PROGRAM

// ---- POUs/LVCP1/PRG_LVCP1_Group4.TcPOU
PROGRAM PRG_LVCP1_Group4
VAR
    // Function Block Instance
    fbContactor: FB_ContactorControl;

    // Contactor 1 IO Structure  
    stContactor_IO: ST_ContactorIO;
    
    // Başlangıç konfigürasyonu için flag
    bContactorInitDone: BOOL := FALSE;
    bCapacitorInitDone: BOOL := FALSE;	
END_VAR



	M_Contactor();
	
	M_Capacitor();

METHOD M_Capacitor : BOOL
VAR
    nGroupIndex : INT;
END_VAR

nGroupIndex := 3;  // Grup 4 için index

IF NOT bCapacitorInitDone THEN
    // Grup 4 değerlerini ata
    GVL_LVCP1.astCompensationGroups[nGroupIndex].rPower := 25.0;
    GVL_LVCP1.astCompensationGroups[nGroupIndex].rVoltage := 450.0;
    GVL_LVCP1.astCompensationGroups[nGroupIndex].nQuantity := 5;
    GVL_LVCP1.astCompensationGroups[nGroupIndex].sTagPrefix := '+EP6-25C1';
    GVL_LVCP1.astCompensationGroups[nGroupIndex].sProductCode := 'ENT.CXD-450-25';
    
    bCapacitorInitDone := TRUE;
END_IF

// Grup 4 aktif durumu
GVL_LVCP1.abGroupActive[nGroupIndex] := stContactor_IO.bFeedback;

M_Capacitor := TRUE;
END_METHOD

METHOD M_Contactor : BOOL
VAR_INPUT
END_VAR
IF NOT bContactorInitDone THEN
    // Konfigürasyon parametreleri
    GVL_LVCP1.stGroup4_ContactorHMI.stConfig.sProjectCode := '+EP6-26K1';
    GVL_LVCP1.stGroup4_ContactorHMI.stConfig.sProductCode := 'SCH LC1G500LSEA';
    GVL_LVCP1.stGroup4_ContactorHMI.stConfig.rRatedCurrent := 500.0;
    GVL_LVCP1.stGroup4_ContactorHMI.stConfig.rRatedVoltage := 1000.0;
    GVL_LVCP1.stGroup4_ContactorHMI.stConfig.nPhaseCount := 3;
    GVL_LVCP1.stGroup4_ContactorHMI.stConfig.tFeedbackDelay := T#500MS;
    GVL_LVCP1.stGroup4_ContactorHMI.stConfig.tWeldedDelay := T#2S;
    GVL_LVCP1.stGroup4_ContactorHMI.stConfig.dwOperationLimit := 100000;
    
    // Başlangıç bakım sayacı
    GVL_LVCP1.stGroup4_ContactorHMI.stStatistics.dwRemainingOperations := GVL_LVCP1.stGroup4_ContactorHMI.stConfig.dwOperationLimit;
    
    bContactorInitDone := TRUE;
END_IF

// Function Block Çağrısı
fbContactor(
    // Fiziksel Girişler
    bFeedback := stContactor_IO.bFeedback,
    bPLCControl := stContactor_IO.bPLCControl,
    
    // Güvenlik Girişleri
    bSafetyLoop := GVL_Alarm.bSafetyLoop,
    bInterlock := FALSE,
    
    // Sistem Girişleri
    bMasterReset := GVL_Alarm.bMasterReset,
    
    // HMI Bağlantısı
    stHMI := GVL_LVCP1.stGroup4_ContactorHMI,
    
    // Fiziksel Çıkış
    bOutput => stContactor_IO.bOutput
);

M_Contactor := TRUE;
END_METHOD

END_PROGRAM

// ---- POUs/LVCP1/PRG_LVCP1_Group5.TcPOU
PROGRAM PRG_LVCP1_Group5
VAR
    // Function Block Instance
    fbContactor: FB_ContactorControl;

    // Contactor 1 IO Structure  
    stContactor_IO: ST_ContactorIO;
    
    // Başlangıç konfigürasyonu için flag
    bContactorInitDone: BOOL := FALSE;
    bCapacitorInitDone: BOOL := FALSE;	
END_VAR



	M_Contactor();
	
	M_Capacitor();

METHOD M_Capacitor : BOOL
VAR
    nGroupIndex : INT;
END_VAR

nGroupIndex := 4;  // Grup 5 için index

IF NOT bCapacitorInitDone THEN
    // Grup 5 değerlerini ata
    GVL_LVCP1.astCompensationGroups[nGroupIndex].rPower := 25.0;
    GVL_LVCP1.astCompensationGroups[nGroupIndex].rVoltage := 450.0;
    GVL_LVCP1.astCompensationGroups[nGroupIndex].nQuantity := 4;
    GVL_LVCP1.astCompensationGroups[nGroupIndex].sTagPrefix := '+EP6-28C1';
    GVL_LVCP1.astCompensationGroups[nGroupIndex].sProductCode := 'ENT.CXD-450-25';
    
    bCapacitorInitDone := TRUE;
END_IF

// Grup 5 aktif durumu
GVL_LVCP1.abGroupActive[nGroupIndex] := stContactor_IO.bFeedback;

M_Capacitor := TRUE;
END_METHOD

METHOD M_Contactor : BOOL
VAR_INPUT
END_VAR
IF NOT bContactorInitDone THEN
    // Konfigürasyon parametreleri
    GVL_LVCP1.stGroup5_ContactorHMI.stConfig.sProjectCode := '+EP6-29K1';
    GVL_LVCP1.stGroup5_ContactorHMI.stConfig.sProductCode := 'SCH LC1G265LSEA';
    GVL_LVCP1.stGroup5_ContactorHMI.stConfig.rRatedCurrent := 265.0;
    GVL_LVCP1.stGroup5_ContactorHMI.stConfig.rRatedVoltage := 1000.0;
    GVL_LVCP1.stGroup5_ContactorHMI.stConfig.nPhaseCount := 3;
    GVL_LVCP1.stGroup5_ContactorHMI.stConfig.tFeedbackDelay := T#500MS;
    GVL_LVCP1.stGroup5_ContactorHMI.stConfig.tWeldedDelay := T#2S;
    GVL_LVCP1.stGroup5_ContactorHMI.stConfig.dwOperationLimit := 100000;
    
    // Başlangıç bakım sayacı
    GVL_LVCP1.stGroup5_ContactorHMI.stStatistics.dwRemainingOperations := GVL_LVCP1.stGroup5_ContactorHMI.stConfig.dwOperationLimit;
    
    bContactorInitDone := TRUE;
END_IF

// Function Block Çağrısı
fbContactor(
    // Fiziksel Girişler
    bFeedback := stContactor_IO.bFeedback,
    bPLCControl := stContactor_IO.bPLCControl,
    
    // Güvenlik Girişleri
    bSafetyLoop := GVL_Alarm.bSafetyLoop,
    bInterlock := FALSE,
    
    // Sistem Girişleri
    bMasterReset := GVL_Alarm.bMasterReset,
    
    // HMI Bağlantısı
    stHMI := GVL_LVCP1.stGroup5_ContactorHMI,
    
    // Fiziksel Çıkış
    bOutput => stContactor_IO.bOutput
);

M_Contactor := TRUE;
END_METHOD

END_PROGRAM

// ---- POUs/LVCP1/PRG_LVCP1_Group6.TcPOU
PROGRAM PRG_LVCP1_Group6
VAR
    // Function Block Instance
    fbContactor: FB_ContactorControl;

    // Contactor 1 IO Structure  
    stContactor_IO: ST_ContactorIO;
    
    // Başlangıç konfigürasyonu için flag
    bContactorInitDone: BOOL := FALSE;
    bCapacitorInitDone: BOOL := FALSE;	
END_VAR



	M_Contactor();
	
	M_Capacitor();

METHOD M_Capacitor : BOOL
VAR
    nGroupIndex : INT;
END_VAR

nGroupIndex := 5;  // Grup 6 için index

IF NOT bCapacitorInitDone THEN
    // Grup 6 değerlerini ata
    GVL_LVCP1.astCompensationGroups[nGroupIndex].rPower := 25.0;
    GVL_LVCP1.astCompensationGroups[nGroupIndex].rVoltage := 450.0;
    GVL_LVCP1.astCompensationGroups[nGroupIndex].nQuantity := 3;
    GVL_LVCP1.astCompensationGroups[nGroupIndex].sTagPrefix := '+EP6-31C1';
    GVL_LVCP1.astCompensationGroups[nGroupIndex].sProductCode := 'ENT.CXD-450-25';
    
    bCapacitorInitDone := TRUE;
END_IF

// Grup 6 aktif durumu
GVL_LVCP1.abGroupActive[nGroupIndex] := stContactor_IO.bFeedback;

M_Capacitor := TRUE;
END_METHOD

METHOD M_Contactor : BOOL
VAR_INPUT
END_VAR
IF NOT bContactorInitDone THEN
    // Konfigürasyon parametreleri
    GVL_LVCP1.stGroup6_ContactorHMI.stConfig.sProjectCode := '+EP6-30K1';
    GVL_LVCP1.stGroup6_ContactorHMI.stConfig.sProductCode := 'SCH LC1G265LSEA';
    GVL_LVCP1.stGroup6_ContactorHMI.stConfig.rRatedCurrent := 265.0;
    GVL_LVCP1.stGroup6_ContactorHMI.stConfig.rRatedVoltage := 1000.0;
    GVL_LVCP1.stGroup6_ContactorHMI.stConfig.nPhaseCount := 3;
    GVL_LVCP1.stGroup6_ContactorHMI.stConfig.tFeedbackDelay := T#500MS;
    GVL_LVCP1.stGroup6_ContactorHMI.stConfig.tWeldedDelay := T#2S;
    GVL_LVCP1.stGroup6_ContactorHMI.stConfig.dwOperationLimit := 100000;
    
    // Başlangıç bakım sayacı
    GVL_LVCP1.stGroup6_ContactorHMI.stStatistics.dwRemainingOperations := GVL_LVCP1.stGroup6_ContactorHMI.stConfig.dwOperationLimit;
    
    bContactorInitDone := TRUE;
END_IF

// Function Block Çağrısı
fbContactor(
    // Fiziksel Girişler
    bFeedback := stContactor_IO.bFeedback,
    bPLCControl := stContactor_IO.bPLCControl,
    
    // Güvenlik Girişleri
    bSafetyLoop := GVL_Alarm.bSafetyLoop,
    bInterlock := FALSE,
    
    // Sistem Girişleri
    bMasterReset := GVL_Alarm.bMasterReset,
    
    // HMI Bağlantısı
    stHMI := GVL_LVCP1.stGroup6_ContactorHMI,
    
    // Fiziksel Çıkış
    bOutput => stContactor_IO.bOutput
);

M_Contactor := TRUE;
END_METHOD

END_PROGRAM

// ---- POUs/LVCP1/PRG_LVCP1_Group7.TcPOU
PROGRAM PRG_LVCP1_Group7
VAR
    // Function Block Instance
    fbContactor: FB_ContactorControl;

    // Contactor 1 IO Structure  
    stContactor_IO: ST_ContactorIO;
    
    // Başlangıç konfigürasyonu için flag
    bContactorInitDone: BOOL := FALSE;
    bCapacitorInitDone: BOOL := FALSE;	
END_VAR



	M_Contactor();
	
	M_Capacitor();

METHOD M_Capacitor : BOOL
VAR
    nGroupIndex : INT;
END_VAR

nGroupIndex := 6;  // Grup 7 için index

IF NOT bCapacitorInitDone THEN
    // Grup 7 değerlerini ata
    GVL_LVCP1.astCompensationGroups[nGroupIndex].rPower := 25.0;
    GVL_LVCP1.astCompensationGroups[nGroupIndex].rVoltage := 450.0;
    GVL_LVCP1.astCompensationGroups[nGroupIndex].nQuantity := 2;
    GVL_LVCP1.astCompensationGroups[nGroupIndex].sTagPrefix := '+EP6-34C1';
    GVL_LVCP1.astCompensationGroups[nGroupIndex].sProductCode := 'ENT.CXD-450-25';
    
    bCapacitorInitDone := TRUE;
END_IF

// Grup 7 aktif durumu
GVL_LVCP1.abGroupActive[nGroupIndex] := stContactor_IO.bFeedback;

M_Capacitor := TRUE;
END_METHOD

METHOD M_Contactor : BOOL
VAR_INPUT
END_VAR
IF NOT bContactorInitDone THEN
    // Konfigürasyon parametreleri
    GVL_LVCP1.stGroup7_ContactorHMI.stConfig.sProjectCode := '+EP6-33K1';
    GVL_LVCP1.stGroup7_ContactorHMI.stConfig.sProductCode := 'SCH LC1G150LSEA';
    GVL_LVCP1.stGroup7_ContactorHMI.stConfig.rRatedCurrent := 150.0;
    GVL_LVCP1.stGroup7_ContactorHMI.stConfig.rRatedVoltage := 1000.0;
    GVL_LVCP1.stGroup7_ContactorHMI.stConfig.nPhaseCount := 3;
    GVL_LVCP1.stGroup7_ContactorHMI.stConfig.tFeedbackDelay := T#500MS;
    GVL_LVCP1.stGroup7_ContactorHMI.stConfig.tWeldedDelay := T#2S;
    GVL_LVCP1.stGroup7_ContactorHMI.stConfig.dwOperationLimit := 100000;
    
    // Başlangıç bakım sayacı
    GVL_LVCP1.stGroup7_ContactorHMI.stStatistics.dwRemainingOperations := GVL_LVCP1.stGroup7_ContactorHMI.stConfig.dwOperationLimit;
    
    bContactorInitDone := TRUE;
END_IF

// Function Block Çağrısı
fbContactor(
    // Fiziksel Girişler
    bFeedback := stContactor_IO.bFeedback,
    bPLCControl := stContactor_IO.bPLCControl,
    
    // Güvenlik Girişleri
    bSafetyLoop := GVL_Alarm.bSafetyLoop,
    bInterlock := FALSE,
    
    // Sistem Girişleri
    bMasterReset := GVL_Alarm.bMasterReset,
    
    // HMI Bağlantısı
    stHMI := GVL_LVCP1.stGroup7_ContactorHMI,
    
    // Fiziksel Çıkış
    bOutput => stContactor_IO.bOutput
);

M_Contactor := TRUE;
END_METHOD

END_PROGRAM

// ---- POUs/LVCP1/PRG_LVCP1_Group8.TcPOU
PROGRAM PRG_LVCP1_Group8
VAR
    // Function Block Instance
    fbContactor: FB_ContactorControl;

    // Contactor 1 IO Structure  
    stContactor_IO: ST_ContactorIO;
    
    // Başlangıç konfigürasyonu için flag
    bContactorInitDone: BOOL := FALSE;
    bCapacitorInitDone: BOOL := FALSE;	
END_VAR



	M_Contactor();
	
	M_Capacitor();

METHOD M_Capacitor : BOOL
VAR
    nGroupIndex : INT;
END_VAR

nGroupIndex := 7;  // Grup 8 için index

IF NOT bCapacitorInitDone THEN
    // Grup 8 değerlerini ata
    GVL_LVCP1.astCompensationGroups[nGroupIndex].rPower := 12.5;
    GVL_LVCP1.astCompensationGroups[nGroupIndex].rVoltage := 450.0;
    GVL_LVCP1.astCompensationGroups[nGroupIndex].nQuantity := 3;
    GVL_LVCP1.astCompensationGroups[nGroupIndex].sTagPrefix := '+EP6-37C1';
    GVL_LVCP1.astCompensationGroups[nGroupIndex].sProductCode := 'ENT.CXD-450-12.5';
    
    bCapacitorInitDone := TRUE;
END_IF

// Grup 8 aktif durumu
GVL_LVCP1.abGroupActive[nGroupIndex] := stContactor_IO.bFeedback;

M_Capacitor := TRUE;
END_METHOD

METHOD M_Contactor : BOOL
VAR_INPUT
END_VAR
IF NOT bContactorInitDone THEN
    // Konfigürasyon parametreleri
    GVL_LVCP1.stGroup8_ContactorHMI.stConfig.sProjectCode := '+EP6-36K1';
    GVL_LVCP1.stGroup8_ContactorHMI.stConfig.sProductCode := 'SCH LC1G115LSEA';
    GVL_LVCP1.stGroup8_ContactorHMI.stConfig.rRatedCurrent := 115.0;
    GVL_LVCP1.stGroup8_ContactorHMI.stConfig.rRatedVoltage := 1000.0;
    GVL_LVCP1.stGroup8_ContactorHMI.stConfig.nPhaseCount := 3;
    GVL_LVCP1.stGroup8_ContactorHMI.stConfig.tFeedbackDelay := T#500MS;
    GVL_LVCP1.stGroup8_ContactorHMI.stConfig.tWeldedDelay := T#2S;
    GVL_LVCP1.stGroup8_ContactorHMI.stConfig.dwOperationLimit := 100000;
    
    // Başlangıç bakım sayacı
    GVL_LVCP1.stGroup8_ContactorHMI.stStatistics.dwRemainingOperations := GVL_LVCP1.stGroup8_ContactorHMI.stConfig.dwOperationLimit;
    
    bContactorInitDone := TRUE;
END_IF

// Function Block Çağrısı
fbContactor(
    // Fiziksel Girişler
    bFeedback := stContactor_IO.bFeedback,
    bPLCControl := stContactor_IO.bPLCControl,
    
    // Güvenlik Girişleri
    bSafetyLoop := GVL_Alarm.bSafetyLoop,
    bInterlock := FALSE,
    
    // Sistem Girişleri
    bMasterReset := GVL_Alarm.bMasterReset,
    
    // HMI Bağlantısı
    stHMI := GVL_LVCP1.stGroup8_ContactorHMI,
    
    // Fiziksel Çıkış
    bOutput => stContactor_IO.bOutput
);

M_Contactor := TRUE;
END_METHOD

END_PROGRAM

// ---- POUs/LVCP1/PRG_LVCP1_Group9.TcPOU
PROGRAM PRG_LVCP1_Group9
VAR
    // Function Block Instance
    fbContactor: FB_ContactorControl;

    // Contactor 1 IO Structure  
    stContactor_IO: ST_ContactorIO;
    
    // Başlangıç konfigürasyonu için flag
    bContactorInitDone: BOOL := FALSE;
    bCapacitorInitDone: BOOL := FALSE;	
END_VAR



	M_Contactor();
	
	M_Capacitor();

METHOD M_Capacitor : BOOL
VAR
    nGroupIndex : INT;
END_VAR

nGroupIndex := 8;  // Grup 9 için index

IF NOT bCapacitorInitDone THEN
    // Grup 9 değerlerini ata
    GVL_LVCP1.astCompensationGroups[nGroupIndex].rPower := 12.5;
    GVL_LVCP1.astCompensationGroups[nGroupIndex].rVoltage := 450.0;
    GVL_LVCP1.astCompensationGroups[nGroupIndex].nQuantity := 2;
    GVL_LVCP1.astCompensationGroups[nGroupIndex].sTagPrefix := '+EP6-40C1';
    GVL_LVCP1.astCompensationGroups[nGroupIndex].sProductCode := 'ENT.CXD-450-12.5';
    
    bCapacitorInitDone := TRUE;
END_IF

// Grup 9 aktif durumu
GVL_LVCP1.abGroupActive[nGroupIndex] := stContactor_IO.bFeedback;

M_Capacitor := TRUE;
END_METHOD

METHOD M_Contactor : BOOL
VAR_INPUT
END_VAR
IF NOT bContactorInitDone THEN
    // Konfigürasyon parametreleri
    GVL_LVCP1.stGroup9_ContactorHMI.stConfig.sProjectCode := '+EP6-39K1';
    GVL_LVCP1.stGroup9_ContactorHMI.stConfig.sProductCode := 'SCH LC1G115LSEA';
    GVL_LVCP1.stGroup9_ContactorHMI.stConfig.rRatedCurrent := 115.0;
    GVL_LVCP1.stGroup9_ContactorHMI.stConfig.rRatedVoltage := 1000.0;
    GVL_LVCP1.stGroup9_ContactorHMI.stConfig.nPhaseCount := 3;
    GVL_LVCP1.stGroup9_ContactorHMI.stConfig.tFeedbackDelay := T#500MS;
    GVL_LVCP1.stGroup9_ContactorHMI.stConfig.tWeldedDelay := T#2S;
    GVL_LVCP1.stGroup9_ContactorHMI.stConfig.dwOperationLimit := 100000;
    
    // Başlangıç bakım sayacı
    GVL_LVCP1.stGroup9_ContactorHMI.stStatistics.dwRemainingOperations := GVL_LVCP1.stGroup9_ContactorHMI.stConfig.dwOperationLimit;
    
    bContactorInitDone := TRUE;
END_IF

// Function Block Çağrısı
fbContactor(
    // Fiziksel Girişler
    bFeedback := stContactor_IO.bFeedback,
    bPLCControl := stContactor_IO.bPLCControl,
    
    // Güvenlik Girişleri
    bSafetyLoop := GVL_Alarm.bSafetyLoop,
    bInterlock := FALSE,
    
    // Sistem Girişleri
    bMasterReset := GVL_Alarm.bMasterReset,
    
    // HMI Bağlantısı
    stHMI := GVL_LVCP1.stGroup9_ContactorHMI,
    
    // Fiziksel Çıkış
    bOutput => stContactor_IO.bOutput
);

M_Contactor := TRUE;
END_METHOD

END_PROGRAM

// ---- POUs/LVCP1/PRG_LVCP1_Group10.TcPOU
PROGRAM PRG_LVCP1_Group10
VAR
    // Function Block Instance
    fbContactor: FB_ContactorControl;

    // Contactor 1 IO Structure  
    stContactor_IO: ST_ContactorIO;
    
    // Başlangıç konfigürasyonu için flag
    bContactorInitDone: BOOL := FALSE;
    bCapacitorInitDone: BOOL := FALSE;	
END_VAR



	M_Contactor();
	
	M_Capacitor();

METHOD M_Capacitor : BOOL
VAR
    nGroupIndex : INT;
END_VAR

nGroupIndex := 9;  // Grup 10 için index

IF NOT bCapacitorInitDone THEN
    // Grup 10 değerlerini ata
    GVL_LVCP1.astCompensationGroups[nGroupIndex].rPower := 12.5;
    GVL_LVCP1.astCompensationGroups[nGroupIndex].rVoltage := 450.0;
    GVL_LVCP1.astCompensationGroups[nGroupIndex].nQuantity := 1;
    GVL_LVCP1.astCompensationGroups[nGroupIndex].sTagPrefix := '+EP6-43C1';
    GVL_LVCP1.astCompensationGroups[nGroupIndex].sProductCode := 'ENT.CXD-450-12.5';
    
    bCapacitorInitDone := TRUE;
END_IF

// Grup 10 aktif durumu
GVL_LVCP1.abGroupActive[nGroupIndex] := stContactor_IO.bFeedback;

M_Capacitor := TRUE;
END_METHOD

METHOD M_Contactor : BOOL
VAR_INPUT
END_VAR
IF NOT bContactorInitDone THEN
    // Konfigürasyon parametreleri
    GVL_LVCP1.stGroup10_ContactorHMI.stConfig.sProjectCode := '+EP6-42K1';
    GVL_LVCP1.stGroup10_ContactorHMI.stConfig.sProductCode := 'SCH LC1G115LSEA';
    GVL_LVCP1.stGroup10_ContactorHMI.stConfig.rRatedCurrent := 115.0;
    GVL_LVCP1.stGroup10_ContactorHMI.stConfig.rRatedVoltage := 1000.0;
    GVL_LVCP1.stGroup10_ContactorHMI.stConfig.nPhaseCount := 3;
    GVL_LVCP1.stGroup10_ContactorHMI.stConfig.tFeedbackDelay := T#500MS;
    GVL_LVCP1.stGroup10_ContactorHMI.stConfig.tWeldedDelay := T#2S;
    GVL_LVCP1.stGroup10_ContactorHMI.stConfig.dwOperationLimit := 100000;
    
    // Başlangıç bakım sayacı
    GVL_LVCP1.stGroup10_ContactorHMI.stStatistics.dwRemainingOperations := GVL_LVCP1.stGroup10_ContactorHMI.stConfig.dwOperationLimit;
    
    bContactorInitDone := TRUE;
END_IF

// Function Block Çağrısı
fbContactor(
    // Fiziksel Girişler
    bFeedback := stContactor_IO.bFeedback,
    bPLCControl := stContactor_IO.bPLCControl,
    
    // Güvenlik Girişleri
    bSafetyLoop := GVL_Alarm.bSafetyLoop,
    bInterlock := FALSE,
    
    // Sistem Girişleri
    bMasterReset := GVL_Alarm.bMasterReset,
    
    // HMI Bağlantısı
    stHMI := GVL_LVCP1.stGroup10_ContactorHMI,
    
    // Fiziksel Çıkış
    bOutput => stContactor_IO.bOutput
);

M_Contactor := TRUE;
END_METHOD

END_PROGRAM

// ---- POUs/LVCP2/PRG_LVCP2.TcPOU
PROGRAM PRG_LVCP2
VAR
END_VAR

	PRG_LVCP2_PowerMeasurement();

	PRG_LVCP2_CompensationCalculate();

	PRG_LVCP2_MainDisconnector();
	
	PRG_LVCP2_Colors();
	
	PRG_LVCP2_Group1();
	
	PRG_LVCP2_Group2();
	
	PRG_LVCP2_Group3();	
	
	PRG_LVCP2_Group4();	

	PRG_LVCP2_Group5();	

	PRG_LVCP2_Group6();	

	PRG_LVCP2_Group7();	

	PRG_LVCP2_Group8();	

	PRG_LVCP2_Group9();	

	PRG_LVCP2_Group10();

END_PROGRAM

// ---- POUs/LVCP2/PRG_LVCP2_PowerMeasurement.TcPOU
PROGRAM PRG_LVCP2_PowerMeasurement
VAR
	// Enerji Yönetimi
	fbEL3453	: FB_EL3453;	
	stEL3453	: stEL3453;
END_VAR


	fbEL3453(pOut := ADR(stEL3453));

END_PROGRAM

